KUKA KRL program: MASTER_MESA_A.src, MASTER_MESA_A.dat

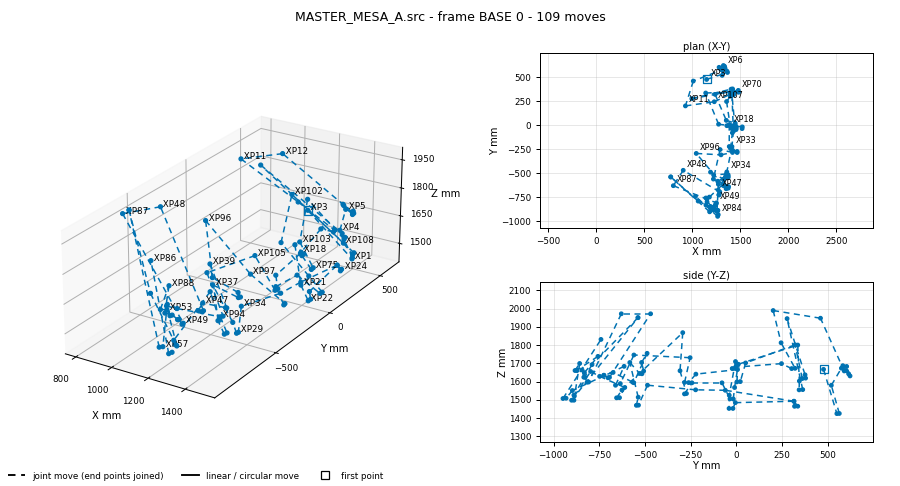
[picture p0: tool path of MASTER_MESA_A.src in frame BASE 0, 109 of 111 moves have a stored position in this frame; points joined in program order, loops and branches not executed]
--- MASTER_MESA_A.src ---
&ACCESS RVP
&REL 294
&PARAM EDITMASK = *
&PARAM TEMPLATE = C:\KRC\Roboter\Template\vorgabe
&PARAM DISKPATH = KRC:\R1\Program\Solda
DEF MASTER_MESA_A( )
;FOLD INI;%{PE}
  ;FOLD BASISTECH INI
    GLOBAL INTERRUPT DECL 3 WHEN $STOPMESS==TRUE DO IR_STOPM ( )
    INTERRUPT ON 3
    BAS (#INITMOV,0 )
  ;ENDFOLD (BASISTECH INI)
  ;FOLD USER INI
    ;Make your modifications here

  ;ENDFOLD (USER INI)
;ENDFOLD (INI)
LOOP
;FOLD PTP HOME Vel=100 % DEFAULT;%{PE}%R 8.3.48,%MKUKATPBASIS,%CMOVE,%VPTP,%P 1:PTP, 2:HOME, 3:, 5:100, 7:DEFAULT
$BWDSTART=FALSE
PDAT_ACT=PDEFAULT
FDAT_ACT=FHOME
BAS(#PTP_PARAMS,100)
$H_POS=XHOME
PTP XHOME
;ENDFOLD

;FOLD PTP P3 Vel=100 % PDAT3 Tool[1]:TOCH Base[0];%{PE}%R 8.3.48,%MKUKATPBASIS,%CMOVE,%VPTP,%P 1:PTP, 2:P3, 3:, 5:100, 7:PDAT3
$BWDSTART=FALSE
PDAT_ACT=PPDAT3
FDAT_ACT=FP3
BAS(#PTP_PARAMS,100)
PTP XP3
;ENDFOLD
;FOLD ; CORDAO 1;%{PE}%R 8.3.48,%MKUKATPBASIS,%CCOMMENT,%VNORMAL,%P 2:CORDAO 1
;ENDFOLD
;FOLD ARCON WDAT1 PTP P1 Vel=30 % PDAT2 Tool[1]:TOCH Base[0] ;%{PE}
;FOLD Parameters ;%{h}
;Params IlfProvider=kukaroboter.arctech.arconptp; Kuka.PointName=P1; Kuka.BlendingEnabled=False; Kuka.MoveDataPtpName=PDAT2; Kuka.VelocityPtp=30; Kuka.MovementParameterFieldEnabled=True; ArcTech.WdatVarName=WDAT1; ArcTech.SeamName=
;ENDFOLD
$BWDSTART = FALSE
PDAT_ACT = PPDAT2
FDAT_ACT = FP1
BAS(#PTP_PARAMS, 30.0)
TRIGGER WHEN DISTANCE = 1 DELAY = ATBg_PreDefinitionTime DO Arc_DefineStrikeParams(3, AS_WDAT1) PRIO = -1
Arc_DefineCpPattern(#OffInAdvance, WV_WDAT1, TRUE)
PTP XP1
Arc_On(1, AS_WDAT1, ATBg_StartErrSetField[1], AW_WDAT1, WV_WDAT1, ATBg_WeldErrSetField[1], #StdArcOn, " ")
Arc_DefineCpPattern(#OnInAdvance, WV_WDAT1, TRUE)
;ENDFOLD
;FOLD ARCOFF WDAT2 LIN P2 CPDAT2 Tool[1]:TOCH Base[0] ;%{PE}
;FOLD Parameters ;%{h}
;Params IlfProvider=kukaroboter.arctech.arcofflin; Kuka.PointName=P2; Kuka.BlendingEnabled=False; Kuka.MoveDataName=CPDAT2;  Kuka.MovementParameterFieldEnabled=True; ArcTech.WdatVarName=WDAT2
;ENDFOLD
$BWDSTART = FALSE
LDAT_ACT = LCPDAT2
FDAT_ACT = FP2
BAS(#CP_PARAMS, ATBg_BAS_VELDefinition)
LIN XP2
Arc_Off(1, AC_WDAT2)
;ENDFOLD
;FOLD PTP P4 Vel=100 % PDAT4 Tool[1]:TOCH Base[0];%{PE}%R 8.3.48,%MKUKATPBASIS,%CMOVE,%VPTP,%P 1:PTP, 2:P4, 3:, 5:100, 7:PDAT4
$BWDSTART=FALSE
PDAT_ACT=PPDAT4
FDAT_ACT=FP4
BAS(#PTP_PARAMS,100)
PTP XP4
;ENDFOLD
;FOLD PTP P5 Vel=100 % PDAT5 Tool[1]:TOCH Base[0];%{PE}%R 8.3.48,%MKUKATPBASIS,%CMOVE,%VPTP,%P 1:PTP, 2:P5, 3:, 5:100, 7:PDAT5
$BWDSTART=FALSE
PDAT_ACT=PPDAT5
FDAT_ACT=FP5
BAS(#PTP_PARAMS,100)
PTP XP5
;ENDFOLD
;FOLD ; CORDAO 2;%{PE}%R 8.3.48,%MKUKATPBASIS,%CCOMMENT,%VNORMAL,%P 2:CORDAO 2
;ENDFOLD
;FOLD ARCON WDAT3 PTP P6 Vel=30 % PDAT6 Tool[1]:TOCH Base[0] ;%{PE}
;FOLD Parameters ;%{h}
;Params IlfProvider=kukaroboter.arctech.arconptp; Kuka.PointName=P6; Kuka.BlendingEnabled=False; Kuka.MoveDataPtpName=PDAT6; Kuka.VelocityPtp=30; Kuka.MovementParameterFieldEnabled=True; ArcTech.WdatVarName=WDAT3; ArcTech.SeamName=
;ENDFOLD
$BWDSTART = FALSE
PDAT_ACT = PPDAT6
FDAT_ACT = FP6
BAS(#PTP_PARAMS, 30.0)
TRIGGER WHEN DISTANCE = 1 DELAY = ATBg_PreDefinitionTime DO Arc_DefineStrikeParams(3, AS_WDAT3) PRIO = -1
Arc_DefineCpPattern(#OffInAdvance, WV_WDAT3, TRUE)
PTP XP6
Arc_On(1, AS_WDAT3, ATBg_StartErrSetField[1], AW_WDAT3, WV_WDAT3, ATBg_WeldErrSetField[1], #StdArcOn, " ")
Arc_DefineCpPattern(#OnInAdvance, WV_WDAT3, TRUE)
;ENDFOLD
;FOLD ARCOFF WDAT4 LIN P7 CPDAT3 Tool[1]:TOCH Base[0] ;%{PE}
;FOLD Parameters ;%{h}
;Params IlfProvider=kukaroboter.arctech.arcofflin; Kuka.PointName=P7; Kuka.BlendingEnabled=False; Kuka.MoveDataName=CPDAT3;  Kuka.MovementParameterFieldEnabled=True; ArcTech.WdatVarName=WDAT4
;ENDFOLD
$BWDSTART = FALSE
LDAT_ACT = LCPDAT3
FDAT_ACT = FP7
BAS(#CP_PARAMS, ATBg_BAS_VELDefinition)
LIN XP7
Arc_Off(1, AC_WDAT4)
;ENDFOLD
;FOLD PTP P8 Vel=100 % PDAT7 Tool[1]:TOCH Base[0];%{PE}%R 8.3.48,%MKUKATPBASIS,%CMOVE,%VPTP,%P 1:PTP, 2:P8, 3:, 5:100, 7:PDAT7
$BWDSTART=FALSE
PDAT_ACT=PPDAT7
FDAT_ACT=FP8
BAS(#PTP_PARAMS,100)
PTP XP8
;ENDFOLD
;FOLD PTP P13 Vel=100 % PDAT11 Tool[1]:TOCH Base[0];%{PE}%R 8.3.48,%MKUKATPBASIS,%CMOVE,%VPTP,%P 1:PTP, 2:P13, 3:, 5:100, 7:PDAT11
$BWDSTART=FALSE
PDAT_ACT=PPDAT11
FDAT_ACT=FP13
BAS(#PTP_PARAMS,100)
PTP XP13
;ENDFOLD
;FOLD ; CORDAO 3;%{PE}%R 8.3.48,%MKUKATPBASIS,%CCOMMENT,%VNORMAL,%P 2:CORDAO 3
;ENDFOLD
;FOLD ARCON WDAT5 PTP P9 Vel=30 % PDAT8 Tool[1]:TOCH Base[0] ;%{PE}
;FOLD Parameters ;%{h}
;Params IlfProvider=kukaroboter.arctech.arconptp; Kuka.PointName=P9; Kuka.BlendingEnabled=False; Kuka.MoveDataPtpName=PDAT8; Kuka.VelocityPtp=30; Kuka.MovementParameterFieldEnabled=True; ArcTech.WdatVarName=WDAT5; ArcTech.SeamName=
;ENDFOLD
$BWDSTART = FALSE
PDAT_ACT = PPDAT8
FDAT_ACT = FP9
BAS(#PTP_PARAMS, 30.0)
TRIGGER WHEN DISTANCE = 1 DELAY = ATBg_PreDefinitionTime DO Arc_DefineStrikeParams(3, AS_WDAT5) PRIO = -1
Arc_DefineCpPattern(#OffInAdvance, WV_WDAT5, TRUE)
PTP XP9
Arc_On(1, AS_WDAT5, ATBg_StartErrSetField[1], AW_WDAT5, WV_WDAT5, ATBg_WeldErrSetField[1], #StdArcOn, " ")
Arc_DefineCpPattern(#OnInAdvance, WV_WDAT5, TRUE)
;ENDFOLD
;FOLD ARCOFF WDAT6 LIN P10 CPDAT4 Tool[1]:TOCH Base[0] ;%{PE}
;FOLD Parameters ;%{h}
;Params IlfProvider=kukaroboter.arctech.arcofflin; Kuka.PointName=P10; Kuka.BlendingEnabled=False; Kuka.MoveDataName=CPDAT4;  Kuka.MovementParameterFieldEnabled=True; ArcTech.WdatVarName=WDAT6
;ENDFOLD
$BWDSTART = FALSE
LDAT_ACT = LCPDAT4
FDAT_ACT = FP10
BAS(#CP_PARAMS, ATBg_BAS_VELDefinition)
LIN XP10
Arc_Off(1, AC_WDAT6)
;ENDFOLD
;FOLD PTP P12 Vel=100 % PDAT10 Tool[1]:TOCH Base[0];%{PE}%R 8.3.48,%MKUKATPBASIS,%CMOVE,%VPTP,%P 1:PTP, 2:P12, 3:, 5:100, 7:PDAT10
$BWDSTART=FALSE
PDAT_ACT=PPDAT10
FDAT_ACT=FP12
BAS(#PTP_PARAMS,100)
PTP XP12
;ENDFOLD
;FOLD PTP P11 Vel=100 % PDAT9 Tool[1]:TOCH Base[0];%{PE}%R 8.3.48,%MKUKATPBASIS,%CMOVE,%VPTP,%P 1:PTP, 2:P11, 3:, 5:100, 7:PDAT9
$BWDSTART=FALSE
PDAT_ACT=PPDAT9
FDAT_ACT=FP11
BAS(#PTP_PARAMS,100)
PTP XP11
;ENDFOLD
;FOLD PTP P107 Vel=100 % PDAT83 Tool[1]:TOCH Base[0];%{PE}%R 8.3.48,%MKUKATPBASIS,%CMOVE,%VPTP,%P 1:PTP, 2:P107, 3:, 5:100, 7:PDAT83
$BWDSTART=FALSE
PDAT_ACT=PPDAT83
FDAT_ACT=FP107
BAS(#PTP_PARAMS,100)
PTP XP107
;ENDFOLD
;FOLD ; CORDAO 4;%{PE}%R 8.3.48,%MKUKATPBASIS,%CCOMMENT,%VNORMAL,%P 2:CORDAO 4
;ENDFOLD
;FOLD ARCON WDAT7 PTP P14 Vel=30 % PDAT12 Tool[1]:TOCH Base[0] ;%{PE}
;FOLD Parameters ;%{h}
;Params IlfProvider=kukaroboter.arctech.arconptp; Kuka.PointName=P14; Kuka.BlendingEnabled=False; Kuka.MoveDataPtpName=PDAT12; Kuka.VelocityPtp=30; Kuka.MovementParameterFieldEnabled=True; ArcTech.WdatVarName=WDAT7; ArcTech.SeamName=
;ENDFOLD
$BWDSTART = FALSE
PDAT_ACT = PPDAT12
FDAT_ACT = FP14
BAS(#PTP_PARAMS, 30.0)
TRIGGER WHEN DISTANCE = 1 DELAY = ATBg_PreDefinitionTime DO Arc_DefineStrikeParams(3, AS_WDAT7) PRIO = -1
Arc_DefineCpPattern(#OffInAdvance, WV_WDAT7, TRUE)
PTP XP14
Arc_On(1, AS_WDAT7, ATBg_StartErrSetField[1], AW_WDAT7, WV_WDAT7, ATBg_WeldErrSetField[1], #StdArcOn, " ")
Arc_DefineCpPattern(#OnInAdvance, WV_WDAT7, TRUE)
;ENDFOLD
;FOLD ARCOFF WDAT8 LIN P15 CPDAT5 Tool[1]:TOCH Base[0] ;%{PE}
;FOLD Parameters ;%{h}
;Params IlfProvider=kukaroboter.arctech.arcofflin; Kuka.PointName=P15; Kuka.BlendingEnabled=False; Kuka.MoveDataName=CPDAT5;  Kuka.MovementParameterFieldEnabled=True; ArcTech.WdatVarName=WDAT8
;ENDFOLD
$BWDSTART = FALSE
LDAT_ACT = LCPDAT5
FDAT_ACT = FP15
BAS(#CP_PARAMS, ATBg_BAS_VELDefinition)
LIN XP15
Arc_Off(1, AC_WDAT8)
;ENDFOLD
;FOLD PTP P19 Vel=100 % PDAT15 Tool[1]:TOCH Base[0];%{PE}%R 8.3.48,%MKUKATPBASIS,%CMOVE,%VPTP,%P 1:PTP, 2:P19, 3:, 5:100, 7:PDAT15
$BWDSTART=FALSE
PDAT_ACT=PPDAT15
FDAT_ACT=FP19
BAS(#PTP_PARAMS,100)
PTP XP19
;ENDFOLD
;FOLD PTP P18 Vel=100 % PDAT14 Tool[1]:TOCH Base[0];%{PE}%R 8.3.48,%MKUKATPBASIS,%CMOVE,%VPTP,%P 1:PTP, 2:P18, 3:, 5:100, 7:PDAT14
$BWDSTART=FALSE
PDAT_ACT=PPDAT14
FDAT_ACT=FP18
BAS(#PTP_PARAMS,100)
PTP XP18
;ENDFOLD
;FOLD ; CORDAO 5;%{PE}%R 8.3.48,%MKUKATPBASIS,%CCOMMENT,%VNORMAL,%P 2:CORDAO 5
;ENDFOLD
;FOLD ARCON WDAT9 PTP P16 Vel=31 % PDAT13 Tool[1]:TOCH Base[0] ;%{PE}
;FOLD Parameters ;%{h}
;Params IlfProvider=kukaroboter.arctech.arconptp; Kuka.PointName=P16; Kuka.BlendingEnabled=False; Kuka.MoveDataPtpName=PDAT13; Kuka.VelocityPtp=31; Kuka.MovementParameterFieldEnabled=True; ArcTech.WdatVarName=WDAT9; ArcTech.SeamName=
;ENDFOLD
$BWDSTART = FALSE
PDAT_ACT = PPDAT13
FDAT_ACT = FP16
BAS(#PTP_PARAMS, 31.0)
TRIGGER WHEN DISTANCE = 1 DELAY = ATBg_PreDefinitionTime DO Arc_DefineStrikeParams(3, AS_WDAT9) PRIO = -1
Arc_DefineCpPattern(#OffInAdvance, WV_WDAT9, TRUE)
PTP XP16
Arc_On(1, AS_WDAT9, ATBg_StartErrSetField[1], AW_WDAT9, WV_WDAT9, ATBg_WeldErrSetField[1], #StdArcOn, " ")
Arc_DefineCpPattern(#OnInAdvance, WV_WDAT9, TRUE)
;ENDFOLD
;FOLD ARCOFF WDAT10 LIN P17 CPDAT6 Tool[1]:TOCH Base[0] ;%{PE}
;FOLD Parameters ;%{h}
;Params IlfProvider=kukaroboter.arctech.arcofflin; Kuka.PointName=P17; Kuka.BlendingEnabled=False; Kuka.MoveDataName=CPDAT6;  Kuka.MovementParameterFieldEnabled=True; ArcTech.WdatVarName=WDAT10
;ENDFOLD
$BWDSTART = FALSE
LDAT_ACT = LCPDAT6
FDAT_ACT = FP17
BAS(#CP_PARAMS, ATBg_BAS_VELDefinition)
LIN XP17
Arc_Off(1, AC_WDAT10)
;ENDFOLD
;FOLD PTP P20 Vel=100 % PDAT16 Tool[1]:TOCH Base[0];%{PE}%R 8.3.48,%MKUKATPBASIS,%CMOVE,%VPTP,%P 1:PTP, 2:P20, 3:, 5:100, 7:PDAT16
$BWDSTART=FALSE
PDAT_ACT=PPDAT16
FDAT_ACT=FP20
BAS(#PTP_PARAMS,100)
PTP XP20
;ENDFOLD
;FOLD PTP P21 Vel=100 % PDAT17 Tool[1]:TOCH Base[0];%{PE}%R 8.3.48,%MKUKATPBASIS,%CMOVE,%VPTP,%P 1:PTP, 2:P21, 3:, 5:100, 7:PDAT17
$BWDSTART=FALSE
PDAT_ACT=PPDAT17
FDAT_ACT=FP21
BAS(#PTP_PARAMS,100)
PTP XP21
;ENDFOLD
;FOLD ; CORDAO 6;%{PE}%R 8.3.48,%MKUKATPBASIS,%CCOMMENT,%VNORMAL,%P 2:CORDAO 6
;ENDFOLD
;FOLD ARCON WDAT11 PTP P22 Vel=30 % PDAT18 Tool[1]:TOCH Base[0] ;%{PE}
;FOLD Parameters ;%{h}
;Params IlfProvider=kukaroboter.arctech.arconptp; Kuka.PointName=P22; Kuka.BlendingEnabled=False; Kuka.MoveDataPtpName=PDAT18; Kuka.VelocityPtp=30; Kuka.MovementParameterFieldEnabled=True; ArcTech.WdatVarName=WDAT11; ArcTech.SeamName=
;ENDFOLD
$BWDSTART = FALSE
PDAT_ACT = PPDAT18
FDAT_ACT = FP22
BAS(#PTP_PARAMS, 30.0)
TRIGGER WHEN DISTANCE = 1 DELAY = ATBg_PreDefinitionTime DO Arc_DefineStrikeParams(3, AS_WDAT11) PRIO = -1
Arc_DefineCpPattern(#OffInAdvance, WV_WDAT11, TRUE)
PTP XP22
Arc_On(1, AS_WDAT11, ATBg_StartErrSetField[1], AW_WDAT11, WV_WDAT11, ATBg_WeldErrSetField[1], #StdArcOn, " ")
Arc_DefineCpPattern(#OnInAdvance, WV_WDAT11, TRUE)
;ENDFOLD
;FOLD ARCOFF WDAT12 LIN P23 CPDAT7 Tool[1]:TOCH Base[0] ;%{PE}
;FOLD Parameters ;%{h}
;Params IlfProvider=kukaroboter.arctech.arcofflin; Kuka.PointName=P23; Kuka.BlendingEnabled=False; Kuka.MoveDataName=CPDAT7;  Kuka.MovementParameterFieldEnabled=True; ArcTech.WdatVarName=WDAT12
;ENDFOLD
$BWDSTART = FALSE
LDAT_ACT = LCPDAT7
FDAT_ACT = FP23
BAS(#CP_PARAMS, ATBg_BAS_VELDefinition)
LIN XP23
Arc_Off(1, AC_WDAT12)
;ENDFOLD
;FOLD PTP P28 Vel=100 % PDAT22 Tool[1]:TOCH Base[0];%{PE}%R 8.3.48,%MKUKATPBASIS,%CMOVE,%VPTP,%P 1:PTP, 2:P28, 3:, 5:100, 7:PDAT22
$BWDSTART=FALSE
PDAT_ACT=PPDAT22
FDAT_ACT=FP28
BAS(#PTP_PARAMS,100)
PTP XP28
;ENDFOLD
;FOLD PTP P27 Vel=100 % PDAT21 Tool[1]:TOCH Base[0];%{PE}%R 8.3.48,%MKUKATPBASIS,%CMOVE,%VPTP,%P 1:PTP, 2:P27, 3:, 5:100, 7:PDAT21
$BWDSTART=FALSE
PDAT_ACT=PPDAT21
FDAT_ACT=FP27
BAS(#PTP_PARAMS,100)
PTP XP27
;ENDFOLD
;FOLD ; CORDAO 7;%{PE}%R 8.3.48,%MKUKATPBASIS,%CCOMMENT,%VNORMAL,%P 2:CORDAO 7
;ENDFOLD
;FOLD ARCON WDAT13 PTP P24 Vel=30 % PDAT19 Tool[1]:TOCH Base[0] ;%{PE}
;FOLD Parameters ;%{h}
;Params IlfProvider=kukaroboter.arctech.arconptp; Kuka.PointName=P24; Kuka.BlendingEnabled=False; Kuka.MoveDataPtpName=PDAT19; Kuka.VelocityPtp=30; Kuka.MovementParameterFieldEnabled=True; ArcTech.WdatVarName=WDAT13; ArcTech.SeamName=
;ENDFOLD
$BWDSTART = FALSE
PDAT_ACT = PPDAT19
FDAT_ACT = FP24
BAS(#PTP_PARAMS, 30.0)
TRIGGER WHEN DISTANCE = 1 DELAY = ATBg_PreDefinitionTime DO Arc_DefineStrikeParams(3, AS_WDAT13) PRIO = -1
Arc_DefineCpPattern(#OffInAdvance, WV_WDAT13, TRUE)
PTP XP24
Arc_On(1, AS_WDAT13, ATBg_StartErrSetField[1], AW_WDAT13, WV_WDAT13, ATBg_WeldErrSetField[1], #StdArcOn, " ")
Arc_DefineCpPattern(#OnInAdvance, WV_WDAT13, TRUE)
;ENDFOLD
;FOLD ARCOFF WDAT14 LIN P25 CPDAT8 Tool[1]:TOCH Base[0] ;%{PE}
;FOLD Parameters ;%{h}
;Params IlfProvider=kukaroboter.arctech.arcofflin; Kuka.PointName=P25; Kuka.BlendingEnabled=False; Kuka.MoveDataName=CPDAT8;  Kuka.MovementParameterFieldEnabled=True; ArcTech.WdatVarName=WDAT14
;ENDFOLD
$BWDSTART = FALSE
LDAT_ACT = LCPDAT8
FDAT_ACT = FP25
BAS(#CP_PARAMS, ATBg_BAS_VELDefinition)
LIN XP25
Arc_Off(1, AC_WDAT14)
;ENDFOLD
;FOLD PTP P26 Vel=100 % PDAT20 Tool[1]:TOCH Base[0];%{PE}%R 8.3.48,%MKUKATPBASIS,%CMOVE,%VPTP,%P 1:PTP, 2:P26, 3:, 5:100, 7:PDAT20
$BWDSTART=FALSE
PDAT_ACT=PPDAT20
FDAT_ACT=FP26
BAS(#PTP_PARAMS,100)
PTP XP26
;ENDFOLD
;FOLD PTP P32 Vel=100 % PDAT25 Tool[1]:TOCH Base[0];%{PE}%R 8.3.48,%MKUKATPBASIS,%CMOVE,%VPTP,%P 1:PTP, 2:P32, 3:, 5:100, 7:PDAT25
$BWDSTART=FALSE
PDAT_ACT=PPDAT25
FDAT_ACT=FP32
BAS(#PTP_PARAMS,100)
PTP XP32
;ENDFOLD
;FOLD PTP P33 Vel=100 % PDAT26 Tool[1]:TOCH Base[0];%{PE}%R 8.3.48,%MKUKATPBASIS,%CMOVE,%VPTP,%P 1:PTP, 2:P33, 3:, 5:100, 7:PDAT26
$BWDSTART=FALSE
PDAT_ACT=PPDAT26
FDAT_ACT=FP33
BAS(#PTP_PARAMS,100)
PTP XP33
;ENDFOLD
;FOLD PTP P34 Vel=100 % PDAT27 Tool[1]:TOCH Base[0];%{PE}%R 8.3.48,%MKUKATPBASIS,%CMOVE,%VPTP,%P 1:PTP, 2:P34, 3:, 5:100, 7:PDAT27
$BWDSTART=FALSE
PDAT_ACT=PPDAT27
FDAT_ACT=FP34
BAS(#PTP_PARAMS,100)
PTP XP34
;ENDFOLD
;FOLD ; CORDAO 8;%{PE}%R 8.3.48,%MKUKATPBASIS,%CCOMMENT,%VNORMAL,%P 2:CORDAO 8
;ENDFOLD
;FOLD ARCON WDAT15 PTP P29 Vel=30 % PDAT23 Tool[1]:TOCH Base[0] ;%{PE}
;FOLD Parameters ;%{h}
;Params IlfProvider=kukaroboter.arctech.arconptp; Kuka.PointName=P29; Kuka.BlendingEnabled=False; Kuka.MoveDataPtpName=PDAT23; Kuka.VelocityPtp=30; Kuka.MovementParameterFieldEnabled=True; ArcTech.WdatVarName=WDAT15; ArcTech.SeamName=
;ENDFOLD
$BWDSTART = FALSE
PDAT_ACT = PPDAT23
FDAT_ACT = FP29
BAS(#PTP_PARAMS, 30.0)
TRIGGER WHEN DISTANCE = 1 DELAY = ATBg_PreDefinitionTime DO Arc_DefineStrikeParams(3, AS_WDAT15) PRIO = -1
Arc_DefineCpPattern(#OffInAdvance, WV_WDAT15, TRUE)
PTP XP29
Arc_On(1, AS_WDAT15, ATBg_StartErrSetField[1], AW_WDAT15, WV_WDAT15, ATBg_WeldErrSetField[1], #StdArcOn, " ")
Arc_DefineCpPattern(#OnInAdvance, WV_WDAT15, TRUE)
;ENDFOLD
;FOLD ARCOFF WDAT16 LIN P30 CPDAT9 Tool[1]:TOCH Base[0] ;%{PE}
;FOLD Parameters ;%{h}
;Params IlfProvider=kukaroboter.arctech.arcofflin; Kuka.PointName=P30; Kuka.BlendingEnabled=False; Kuka.MoveDataName=CPDAT9;  Kuka.MovementParameterFieldEnabled=True; ArcTech.WdatVarName=WDAT16
;ENDFOLD
$BWDSTART = FALSE
LDAT_ACT = LCPDAT9
FDAT_ACT = FP30
BAS(#CP_PARAMS, ATBg_BAS_VELDefinition)
LIN XP30
Arc_Off(1, AC_WDAT16)
;ENDFOLD
;FOLD PTP P31 Vel=100 % PDAT24 Tool[1]:TOCH Base[0];%{PE}%R 8.3.48,%MKUKATPBASIS,%CMOVE,%VPTP,%P 1:PTP, 2:P31, 3:, 5:100, 7:PDAT24
$BWDSTART=FALSE
PDAT_ACT=PPDAT24
FDAT_ACT=FP31
BAS(#PTP_PARAMS,100)
PTP XP31
;ENDFOLD
;FOLD PTP P37 Vel=100 % PDAT29 Tool[1]:TOCH Base[0];%{PE}%R 8.3.48,%MKUKATPBASIS,%CMOVE,%VPTP,%P 1:PTP, 2:P37, 3:, 5:100, 7:PDAT29
$BWDSTART=FALSE
PDAT_ACT=PPDAT29
FDAT_ACT=FP37
BAS(#PTP_PARAMS,100)
PTP XP37
;ENDFOLD
;FOLD ; CORDAO 9;%{PE}%R 8.3.48,%MKUKATPBASIS,%CCOMMENT,%VNORMAL,%P 2:CORDAO 9
;ENDFOLD
;FOLD ARCON WDAT17 PTP P35 Vel=30 % PDAT28 Tool[1]:TOCH Base[0] ;%{PE}
;FOLD Parameters ;%{h}
;Params IlfProvider=kukaroboter.arctech.arconptp; Kuka.PointName=P35; Kuka.BlendingEnabled=False; Kuka.MoveDataPtpName=PDAT28; Kuka.VelocityPtp=30; Kuka.MovementParameterFieldEnabled=True; ArcTech.WdatVarName=WDAT17; ArcTech.SeamName=
;ENDFOLD
$BWDSTART = FALSE
PDAT_ACT = PPDAT28
FDAT_ACT = FP35
BAS(#PTP_PARAMS, 30.0)
TRIGGER WHEN DISTANCE = 1 DELAY = ATBg_PreDefinitionTime DO Arc_DefineStrikeParams(3, AS_WDAT17) PRIO = -1
Arc_DefineCpPattern(#OffInAdvance, WV_WDAT17, TRUE)
PTP XP35
Arc_On(1, AS_WDAT17, ATBg_StartErrSetField[1], AW_WDAT17, WV_WDAT17, ATBg_WeldErrSetField[1], #StdArcOn, " ")
Arc_DefineCpPattern(#OnInAdvance, WV_WDAT17, TRUE)
;ENDFOLD
;FOLD ARCOFF WDAT18 LIN P36 CPDAT10 Tool[1]:TOCH Base[0] ;%{PE}
;FOLD Parameters ;%{h}
;Params IlfProvider=kukaroboter.arctech.arcofflin; Kuka.PointName=P36; Kuka.BlendingEnabled=False; Kuka.MoveDataName=CPDAT10;  Kuka.MovementParameterFieldEnabled=True; ArcTech.WdatVarName=WDAT18
;ENDFOLD
$BWDSTART = FALSE
LDAT_ACT = LCPDAT10
FDAT_ACT = FP36
BAS(#CP_PARAMS, ATBg_BAS_VELDefinition)
LIN XP36
Arc_Off(1, AC_WDAT18)
;ENDFOLD
;FOLD PTP P38 Vel=100 % PDAT30 Tool[1]:TOCH Base[0];%{PE}%R 8.3.48,%MKUKATPBASIS,%CMOVE,%VPTP,%P 1:PTP, 2:P38, 3:, 5:100, 7:PDAT30
$BWDSTART=FALSE
PDAT_ACT=PPDAT30
FDAT_ACT=FP38
BAS(#PTP_PARAMS,100)
PTP XP38
;ENDFOLD
;FOLD PTP P40 Vel=100 % PDAT32 Tool[1]:TOCH Base[0];%{PE}%R 8.3.48,%MKUKATPBASIS,%CMOVE,%VPTP,%P 1:PTP, 2:P40, 3:, 5:100, 7:PDAT32
$BWDSTART=FALSE
PDAT_ACT=PPDAT32
FDAT_ACT=FP40
BAS(#PTP_PARAMS,100)
PTP XP40
;ENDFOLD
;FOLD PTP P39 Vel=100 % PDAT31 Tool[1]:TOCH Base[0];%{PE}%R 8.3.48,%MKUKATPBASIS,%CMOVE,%VPTP,%P 1:PTP, 2:P39, 3:, 5:100, 7:PDAT31
$BWDSTART=FALSE
PDAT_ACT=PPDAT31
FDAT_ACT=FP39
BAS(#PTP_PARAMS,100)
PTP XP39
;ENDFOLD
;FOLD ; CORDAO 10;%{PE}%R 8.3.48,%MKUKATPBASIS,%CCOMMENT,%VNORMAL,%P 2:CORDAO 10
;ENDFOLD
;FOLD ARCON WDAT19 PTP P41 Vel=30 % PDAT33 Tool[1]:TOCH Base[0] ;%{PE}
;FOLD Parameters ;%{h}
;Params IlfProvider=kukaroboter.arctech.arconptp; Kuka.PointName=P41; Kuka.BlendingEnabled=False; Kuka.MoveDataPtpName=PDAT33; Kuka.VelocityPtp=30; Kuka.MovementParameterFieldEnabled=True; ArcTech.WdatVarName=WDAT19; ArcTech.SeamName=
;ENDFOLD
$BWDSTART = FALSE
PDAT_ACT = PPDAT33
FDAT_ACT = FP41
BAS(#PTP_PARAMS, 30.0)
TRIGGER WHEN DISTANCE = 1 DELAY = ATBg_PreDefinitionTime DO Arc_DefineStrikeParams(3, AS_WDAT19) PRIO = -1
Arc_DefineCpPattern(#OffInAdvance, WV_WDAT19, TRUE)
PTP XP41
Arc_On(1, AS_WDAT19, ATBg_StartErrSetField[1], AW_WDAT19, WV_WDAT19, ATBg_WeldErrSetField[1], #StdArcOn, " ")
Arc_DefineCpPattern(#OnInAdvance, WV_WDAT19, TRUE)
;ENDFOLD
;FOLD ARCOFF WDAT20 LIN P42 CPDAT11 Tool[1]:TOCH Base[0] ;%{PE}
;FOLD Parameters ;%{h}
;Params IlfProvider=kukaroboter.arctech.arcofflin; Kuka.PointName=P42; Kuka.BlendingEnabled=False; Kuka.MoveDataName=CPDAT11;  Kuka.MovementParameterFieldEnabled=True; ArcTech.WdatVarName=WDAT20
;ENDFOLD
$BWDSTART = FALSE
LDAT_ACT = LCPDAT11
FDAT_ACT = FP42
BAS(#CP_PARAMS, ATBg_BAS_VELDefinition)
LIN XP42
Arc_Off(1, AC_WDAT20)
;ENDFOLD
;FOLD PTP P47 Vel=100 % PDAT36 Tool[1]:TOCH Base[0];%{PE}%R 8.3.48,%MKUKATPBASIS,%CMOVE,%VPTP,%P 1:PTP, 2:P47, 3:, 5:100, 7:PDAT36
$BWDSTART=FALSE
PDAT_ACT=PPDAT36
FDAT_ACT=FP47
BAS(#PTP_PARAMS,100)
PTP XP47
;ENDFOLD
;FOLD ; CORDAO 11;%{PE}%R 8.3.48,%MKUKATPBASIS,%CCOMMENT,%VNORMAL,%P 2:CORDAO 11
;ENDFOLD
;FOLD ARCON WDAT21 PTP P43 Vel=30 % PDAT34 Tool[1]:TOCH Base[0] ;%{PE}
;FOLD Parameters ;%{h}
;Params IlfProvider=kukaroboter.arctech.arconptp; Kuka.PointName=P43; Kuka.BlendingEnabled=False; Kuka.MoveDataPtpName=PDAT34; Kuka.VelocityPtp=30; Kuka.MovementParameterFieldEnabled=True; ArcTech.WdatVarName=WDAT21; ArcTech.SeamName=
;ENDFOLD
$BWDSTART = FALSE
PDAT_ACT = PPDAT34
FDAT_ACT = FP43
BAS(#PTP_PARAMS, 30.0)
TRIGGER WHEN DISTANCE = 1 DELAY = ATBg_PreDefinitionTime DO Arc_DefineStrikeParams(3, AS_WDAT21) PRIO = -1
Arc_DefineCpPattern(#OffInAdvance, WV_WDAT21, TRUE)
PTP XP43
Arc_On(1, AS_WDAT21, ATBg_StartErrSetField[1], AW_WDAT21, WV_WDAT21, ATBg_WeldErrSetField[1], #StdArcOn, " ")
Arc_DefineCpPattern(#OnInAdvance, WV_WDAT21, TRUE)
;ENDFOLD
;FOLD ARCOFF WDAT22 LIN P44 CPDAT12 Tool[1]:TOCH Base[0] ;%{PE}
;FOLD Parameters ;%{h}
;Params IlfProvider=kukaroboter.arctech.arcofflin; Kuka.PointName=P44; Kuka.BlendingEnabled=False; Kuka.MoveDataName=CPDAT12;  Kuka.MovementParameterFieldEnabled=True; ArcTech.WdatVarName=WDAT22
;ENDFOLD
$BWDSTART = FALSE
LDAT_ACT = LCPDAT12
FDAT_ACT = FP44
BAS(#CP_PARAMS, ATBg_BAS_VELDefinition)
LIN XP44
Arc_Off(1, AC_WDAT22)
;ENDFOLD
;FOLD ; CORDAO 12;%{PE}%R 8.3.48,%MKUKATPBASIS,%CCOMMENT,%VNORMAL,%P 2:CORDAO 12
;ENDFOLD
;FOLD ARCON WDAT23 PTP P45 Vel=30 % PDAT35 Tool[1]:TOCH Base[0] ;%{PE}
;FOLD Parameters ;%{h}
;Params IlfProvider=kukaroboter.arctech.arconptp; Kuka.PointName=P45; Kuka.BlendingEnabled=False; Kuka.MoveDataPtpName=PDAT35; Kuka.VelocityPtp=30; Kuka.MovementParameterFieldEnabled=True; ArcTech.WdatVarName=WDAT23; ArcTech.SeamName=
;ENDFOLD
$BWDSTART = FALSE
PDAT_ACT = PPDAT35
FDAT_ACT = FP45
BAS(#PTP_PARAMS, 30.0)
TRIGGER WHEN DISTANCE = 1 DELAY = ATBg_PreDefinitionTime DO Arc_DefineStrikeParams(1, AS_WDAT23) PRIO = -1
Arc_DefineCpPattern(#OffInAdvance, WV_WDAT23, TRUE)
PTP XP45
Arc_On(1, AS_WDAT23, ATBg_StartErrSetField[1], AW_WDAT23, WV_WDAT23, ATBg_WeldErrSetField[1], #StdArcOn, " ")
Arc_DefineCpPattern(#OnInAdvance, WV_WDAT23, TRUE)
;ENDFOLD
;FOLD ARCOFF WDAT24 LIN P46 CPDAT13 Tool[1]:TOCH Base[0] ;%{PE}
;FOLD Parameters ;%{h}
;Params IlfProvider=kukaroboter.arctech.arcofflin; Kuka.PointName=P46; Kuka.BlendingEnabled=False; Kuka.MoveDataName=CPDAT13;  Kuka.MovementParameterFieldEnabled=True; ArcTech.WdatVarName=WDAT24
;ENDFOLD
$BWDSTART = FALSE
LDAT_ACT = LCPDAT13
FDAT_ACT = FP46
BAS(#CP_PARAMS, ATBg_BAS_VELDefinition)
LIN XP46
Arc_Off(1, AC_WDAT24)
;ENDFOLD
;FOLD PTP P48 Vel=100 % PDAT37 Tool[1]:TOCH Base[0];%{PE}%R 8.3.48,%MKUKATPBASIS,%CMOVE,%VPTP,%P 1:PTP, 2:P48, 3:, 5:100, 7:PDAT37
$BWDSTART=FALSE
PDAT_ACT=PPDAT37
FDAT_ACT=FP48
BAS(#PTP_PARAMS,100)
PTP XP48
;ENDFOLD
;FOLD PTP P87 Vel=100 % PDAT62 Tool[1]:TOCH Base[0];%{PE}%R 8.3.48,%MKUKATPBASIS,%CMOVE,%VPTP,%P 1:PTP, 2:P87, 3:, 5:100, 7:PDAT62
$BWDSTART=FALSE
PDAT_ACT=PPDAT62
FDAT_ACT=FP87
BAS(#PTP_PARAMS,100)
PTP XP87
;ENDFOLD
;FOLD ; CORDAO 13;%{PE}%R 8.3.48,%MKUKATPBASIS,%CCOMMENT,%VNORMAL,%P 2:CORDAO 13
;ENDFOLD
;FOLD ARCON WDAT25 PTP P49 Vel=30 % PDAT38 Tool[1]:TOCH Base[0] ;%{PE}
;FOLD Parameters ;%{h}
;Params IlfProvider=kukaroboter.arctech.arconptp; Kuka.PointName=P49; Kuka.BlendingEnabled=False; Kuka.MoveDataPtpName=PDAT38; Kuka.VelocityPtp=30; Kuka.MovementParameterFieldEnabled=True; ArcTech.WdatVarName=WDAT25; ArcTech.SeamName=
;ENDFOLD
$BWDSTART = FALSE
PDAT_ACT = PPDAT38
FDAT_ACT = FP49
BAS(#PTP_PARAMS, 30.0)
TRIGGER WHEN DISTANCE = 1 DELAY = ATBg_PreDefinitionTime DO Arc_DefineStrikeParams(3, AS_WDAT25) PRIO = -1
Arc_DefineCpPattern(#OffInAdvance, WV_WDAT25, TRUE)
PTP XP49
Arc_On(1, AS_WDAT25, ATBg_StartErrSetField[1], AW_WDAT25, WV_WDAT25, ATBg_WeldErrSetField[1], #StdArcOn, " ")
Arc_DefineCpPattern(#OnInAdvance, WV_WDAT25, TRUE)
;ENDFOLD
;FOLD ARCOFF WDAT26 LIN P50 CPDAT14 Tool[1]:TOCH Base[0] ;%{PE}
;FOLD Parameters ;%{h}
;Params IlfProvider=kukaroboter.arctech.arcofflin; Kuka.PointName=P50; Kuka.BlendingEnabled=False; Kuka.MoveDataName=CPDAT14;  Kuka.MovementParameterFieldEnabled=True; ArcTech.WdatVarName=WDAT26
;ENDFOLD
$BWDSTART = FALSE
LDAT_ACT = LCPDAT14
FDAT_ACT = FP50
BAS(#CP_PARAMS, ATBg_BAS_VELDefinition)
LIN XP50
Arc_Off(1, AC_WDAT26)
;ENDFOLD
;FOLD ; CORDAO 14;%{PE}%R 8.3.48,%MKUKATPBASIS,%CCOMMENT,%VNORMAL,%P 2:CORDAO 14
;ENDFOLD
;FOLD ARCON WDAT27 PTP P51 Vel=30 % PDAT39 Tool[1]:TOCH Base[0] ;%{PE}
;FOLD Parameters ;%{h}
;Params IlfProvider=kukaroboter.arctech.arconptp; Kuka.PointName=P51; Kuka.BlendingEnabled=False; Kuka.MoveDataPtpName=PDAT39; Kuka.VelocityPtp=30; Kuka.MovementParameterFieldEnabled=True; ArcTech.WdatVarName=WDAT27; ArcTech.SeamName=
;ENDFOLD
$BWDSTART = FALSE
PDAT_ACT = PPDAT39
FDAT_ACT = FP51
BAS(#PTP_PARAMS, 30.0)
TRIGGER WHEN DISTANCE = 1 DELAY = ATBg_PreDefinitionTime DO Arc_DefineStrikeParams(3, AS_WDAT27) PRIO = -1
Arc_DefineCpPattern(#OffInAdvance, WV_WDAT27, TRUE)
PTP XP51
Arc_On(1, AS_WDAT27, ATBg_StartErrSetField[1], AW_WDAT27, WV_WDAT27, ATBg_WeldErrSetField[1], #StdArcOn, " ")
Arc_DefineCpPattern(#OnInAdvance, WV_WDAT27, TRUE)
;ENDFOLD
;FOLD ARCOFF WDAT28 LIN P52 CPDAT15 Tool[1]:TOCH Base[0] ;%{PE}
;FOLD Parameters ;%{h}
;Params IlfProvider=kukaroboter.arctech.arcofflin; Kuka.PointName=P52; Kuka.BlendingEnabled=False; Kuka.MoveDataName=CPDAT15;  Kuka.MovementParameterFieldEnabled=True; ArcTech.WdatVarName=WDAT28
;ENDFOLD
$BWDSTART = FALSE
LDAT_ACT = LCPDAT15
FDAT_ACT = FP52
BAS(#CP_PARAMS, ATBg_BAS_VELDefinition)
LIN XP52
Arc_Off(1, AC_WDAT28)
;ENDFOLD
;FOLD PTP P53 Vel=100 % PDAT40 Tool[1]:TOCH Base[0];%{PE}%R 8.3.48,%MKUKATPBASIS,%CMOVE,%VPTP,%P 1:PTP, 2:P53, 3:, 5:100, 7:PDAT40
$BWDSTART=FALSE
PDAT_ACT=PPDAT40
FDAT_ACT=FP53
BAS(#PTP_PARAMS,100)
PTP XP53
;ENDFOLD
;FOLD PTP P89 Vel=100 % PDAT64 Tool[1]:TOCH Base[0];%{PE}%R 8.3.48,%MKUKATPBASIS,%CMOVE,%VPTP,%P 1:PTP, 2:P89, 3:, 5:100, 7:PDAT64
$BWDSTART=FALSE
PDAT_ACT=PPDAT64
FDAT_ACT=FP89
BAS(#PTP_PARAMS,100)
PTP XP89
;ENDFOLD
;FOLD PTP P88 Vel=100 % PDAT63 Tool[1]:TOCH Base[0];%{PE}%R 8.3.48,%MKUKATPBASIS,%CMOVE,%VPTP,%P 1:PTP, 2:P88, 3:, 5:100, 7:PDAT63
$BWDSTART=FALSE
PDAT_ACT=PPDAT63
FDAT_ACT=FP88
BAS(#PTP_PARAMS,100)
PTP XP88
;ENDFOLD
;FOLD PTP P90 Vel=100 % PDAT65 Tool[1]:TOCH Base[0];%{PE}%R 8.3.48,%MKUKATPBASIS,%CMOVE,%VPTP,%P 1:PTP, 2:P90, 3:, 5:100, 7:PDAT65
$BWDSTART=FALSE
PDAT_ACT=PPDAT65
FDAT_ACT=FP90
BAS(#PTP_PARAMS,100)
PTP XP90
;ENDFOLD
;FOLD ; CORDAO 15;%{PE}%R 8.3.48,%MKUKATPBASIS,%CCOMMENT,%VNORMAL,%P 2:CORDAO 15
;ENDFOLD
;FOLD ARCON WDAT29 PTP P54 Vel=30 % PDAT41 Tool[1]:TOCH Base[0] ;%{PE}
;FOLD Parameters ;%{h}
;Params IlfProvider=kukaroboter.arctech.arconptp; Kuka.PointName=P54; Kuka.BlendingEnabled=False; Kuka.MoveDataPtpName=PDAT41; Kuka.VelocityPtp=30; Kuka.MovementParameterFieldEnabled=True; ArcTech.WdatVarName=WDAT29; ArcTech.SeamName=
;ENDFOLD
$BWDSTART = FALSE
PDAT_ACT = PPDAT41
FDAT_ACT = FP54
BAS(#PTP_PARAMS, 30.0)
TRIGGER WHEN DISTANCE = 1 DELAY = ATBg_PreDefinitionTime DO Arc_DefineStrikeParams(3, AS_WDAT29) PRIO = -1
Arc_DefineCpPattern(#OffInAdvance, WV_WDAT29, TRUE)
PTP XP54
Arc_On(1, AS_WDAT29, ATBg_StartErrSetField[1], AW_WDAT29, WV_WDAT29, ATBg_WeldErrSetField[1], #StdArcOn, " ")
Arc_DefineCpPattern(#OnInAdvance, WV_WDAT29, TRUE)
;ENDFOLD
;FOLD ARCOFF WDAT30 LIN P55 CPDAT16 Tool[1]:TOCH Base[0] ;%{PE}
;FOLD Parameters ;%{h}
;Params IlfProvider=kukaroboter.arctech.arcofflin; Kuka.PointName=P55; Kuka.BlendingEnabled=False; Kuka.MoveDataName=CPDAT16;  Kuka.MovementParameterFieldEnabled=True; ArcTech.WdatVarName=WDAT30
;ENDFOLD
$BWDSTART = FALSE
LDAT_ACT = LCPDAT16
FDAT_ACT = FP55
BAS(#CP_PARAMS, ATBg_BAS_VELDefinition)
LIN XP55
Arc_Off(1, AC_WDAT30)
;ENDFOLD
;FOLD PTP P56 Vel=100 % PDAT42 Tool[1]:TOCH Base[0];%{PE}%R 8.3.48,%MKUKATPBASIS,%CMOVE,%VPTP,%P 1:PTP, 2:P56, 3:, 5:100, 7:PDAT42
$BWDSTART=FALSE
PDAT_ACT=PPDAT42
FDAT_ACT=FP56
BAS(#PTP_PARAMS,100)
PTP XP56
;ENDFOLD
;FOLD ; CORDAO 16;%{PE}%R 8.3.48,%MKUKATPBASIS,%CCOMMENT,%VNORMAL,%P 2:CORDAO 16
;ENDFOLD
;FOLD ARCON WDAT31 PTP P57 Vel=30 % PDAT43 Tool[1]:TOCH Base[0] ;%{PE}
;FOLD Parameters ;%{h}
;Params IlfProvider=kukaroboter.arctech.arconptp; Kuka.PointName=P57; Kuka.BlendingEnabled=False; Kuka.MoveDataPtpName=PDAT43; Kuka.VelocityPtp=30; Kuka.MovementParameterFieldEnabled=True; ArcTech.WdatVarName=WDAT31; ArcTech.SeamName=
;ENDFOLD
$BWDSTART = FALSE
PDAT_ACT = PPDAT43
FDAT_ACT = FP57
BAS(#PTP_PARAMS, 30.0)
TRIGGER WHEN DISTANCE = 1 DELAY = ATBg_PreDefinitionTime DO Arc_DefineStrikeParams(3, AS_WDAT31) PRIO = -1
Arc_DefineCpPattern(#OffInAdvance, WV_WDAT31, TRUE)
PTP XP57
Arc_On(1, AS_WDAT31, ATBg_StartErrSetField[1], AW_WDAT31, WV_WDAT31, ATBg_WeldErrSetField[1], #StdArcOn, " ")
Arc_DefineCpPattern(#OnInAdvance, WV_WDAT31, TRUE)
;ENDFOLD
;FOLD ARCOFF WDAT32 LIN P58 CPDAT17 Tool[1]:TOCH Base[0] ;%{PE}
;FOLD Parameters ;%{h}
;Params IlfProvider=kukaroboter.arctech.arcofflin; Kuka.PointName=P58; Kuka.BlendingEnabled=False; Kuka.MoveDataName=CPDAT17;  Kuka.MovementParameterFieldEnabled=True; ArcTech.WdatVarName=WDAT32
;ENDFOLD
$BWDSTART = FALSE
LDAT_ACT = LCPDAT17
FDAT_ACT = FP58
BAS(#CP_PARAMS, ATBg_BAS_VELDefinition)
LIN XP58
Arc_Off(1, AC_WDAT32)
;ENDFOLD
;FOLD PTP P59 Vel=100 % PDAT44 Tool[1]:TOCH Base[0];%{PE}%R 8.3.48,%MKUKATPBASIS,%CMOVE,%VPTP,%P 1:PTP, 2:P59, 3:, 5:100, 7:PDAT44
$BWDSTART=FALSE
PDAT_ACT=PPDAT44
FDAT_ACT=FP59
BAS(#PTP_PARAMS,100)
PTP XP59
;ENDFOLD
;FOLD PTP P60 Vel=100 % PDAT45 Tool[1]:TOCH Base[0];%{PE}%R 8.3.48,%MKUKATPBASIS,%CMOVE,%VPTP,%P 1:PTP, 2:P60, 3:, 5:100, 7:PDAT45
$BWDSTART=FALSE
PDAT_ACT=PPDAT45
FDAT_ACT=FP60
BAS(#PTP_PARAMS,100)
PTP XP60
;ENDFOLD
;FOLD PTP P91 Vel=100 % PDAT67 Tool[1]:TOCH Base[0];%{PE}%R 8.3.48,%MKUKATPBASIS,%CMOVE,%VPTP,%P 1:PTP, 2:P91, 3:, 5:100, 7:PDAT67
$BWDSTART=FALSE
PDAT_ACT=PPDAT67
FDAT_ACT=FP91
BAS(#PTP_PARAMS,100)
PTP XP91
;ENDFOLD
;FOLD ; CORDAO 17;%{PE}%R 8.3.48,%MKUKATPBASIS,%CCOMMENT,%VNORMAL,%P 2:CORDAO 17
;ENDFOLD
;FOLD ARCON WDAT33 PTP P61 Vel=30 % PDAT66 Tool[1]:TOCH Base[0] ;%{PE}
;FOLD Parameters ;%{h}
;Params IlfProvider=kukaroboter.arctech.arconptp; Kuka.PointName=P61; Kuka.BlendingEnabled=False; Kuka.MoveDataPtpName=PDAT66; Kuka.VelocityPtp=30; Kuka.MovementParameterFieldEnabled=True; ArcTech.WdatVarName=WDAT33; ArcTech.SeamName=
;ENDFOLD
$BWDSTART = FALSE
PDAT_ACT = PPDAT66
FDAT_ACT = FP61
BAS(#PTP_PARAMS, 30.0)
TRIGGER WHEN DISTANCE = 1 DELAY = ATBg_PreDefinitionTime DO Arc_DefineStrikeParams(3, AS_WDAT33) PRIO = -1
Arc_DefineCpPattern(#OffInAdvance, WV_WDAT33, TRUE)
PTP XP61
Arc_On(1, AS_WDAT33, ATBg_StartErrSetField[1], AW_WDAT33, WV_WDAT33, ATBg_WeldErrSetField[1], #StdArcOn, " ")
Arc_DefineCpPattern(#OnInAdvance, WV_WDAT33, TRUE)
;ENDFOLD
;FOLD ARCOFF WDAT34 LIN P62 CPDAT18 Tool[1]:TOCH Base[0] ;%{PE}
;FOLD Parameters ;%{h}
;Params IlfProvider=kukaroboter.arctech.arcofflin; Kuka.PointName=P62; Kuka.BlendingEnabled=False; Kuka.MoveDataName=CPDAT18;  Kuka.MovementParameterFieldEnabled=True; ArcTech.WdatVarName=WDAT34
;ENDFOLD
$BWDSTART = FALSE
LDAT_ACT = LCPDAT18
FDAT_ACT = FP62
BAS(#CP_PARAMS, ATBg_BAS_VELDefinition)
LIN XP62
Arc_Off(1, AC_WDAT34)
;ENDFOLD
;FOLD PTP P92 Vel=100 % PDAT68 Tool[1]:TOCH Base[0];%{PE}%R 8.3.48,%MKUKATPBASIS,%CMOVE,%VPTP,%P 1:PTP, 2:P92, 3:, 5:100, 7:PDAT68
$BWDSTART=FALSE
PDAT_ACT=PPDAT68
FDAT_ACT=FP92
BAS(#PTP_PARAMS,100)
PTP XP92
;ENDFOLD
;FOLD PTP P93 Vel=100 % PDAT69 Tool[1]:TOCH Base[0];%{PE}%R 8.3.48,%MKUKATPBASIS,%CMOVE,%VPTP,%P 1:PTP, 2:P93, 3:, 5:100, 7:PDAT69
$BWDSTART=FALSE
PDAT_ACT=PPDAT69
FDAT_ACT=FP93
BAS(#PTP_PARAMS,100)
PTP XP93
;ENDFOLD
;FOLD PTP P94 Vel=100 % PDAT70 Tool[1]:TOCH Base[0];%{PE}%R 8.3.48,%MKUKATPBASIS,%CMOVE,%VPTP,%P 1:PTP, 2:P94, 3:, 5:100, 7:PDAT70
$BWDSTART=FALSE
PDAT_ACT=PPDAT70
FDAT_ACT=FP94
BAS(#PTP_PARAMS,100)
PTP XP94
;ENDFOLD
;FOLD ; CORDAO 18;%{PE}%R 8.3.48,%MKUKATPBASIS,%CCOMMENT,%VNORMAL,%P 2:CORDAO 18
;ENDFOLD
;FOLD ARCON WDAT35 PTP P63 Vel=30 % PDAT47 Tool[1]:TOCH Base[0] ;%{PE}
;FOLD Parameters ;%{h}
;Params IlfProvider=kukaroboter.arctech.arconptp; Kuka.PointName=P63; Kuka.BlendingEnabled=False; Kuka.MoveDataPtpName=PDAT47; Kuka.VelocityPtp=30; Kuka.MovementParameterFieldEnabled=True; ArcTech.WdatVarName=WDAT35; ArcTech.SeamName=
;ENDFOLD
$BWDSTART = FALSE
PDAT_ACT = PPDAT47
FDAT_ACT = FP63
BAS(#PTP_PARAMS, 30.0)
TRIGGER WHEN DISTANCE = 1 DELAY = ATBg_PreDefinitionTime DO Arc_DefineStrikeParams(3, AS_WDAT35) PRIO = -1
Arc_DefineCpPattern(#OffInAdvance, WV_WDAT35, TRUE)
PTP XP63
Arc_On(1, AS_WDAT35, ATBg_StartErrSetField[1], AW_WDAT35, WV_WDAT35, ATBg_WeldErrSetField[1], #StdArcOn, " ")
Arc_DefineCpPattern(#OnInAdvance, WV_WDAT35, TRUE)
;ENDFOLD
;FOLD ARCOFF WDAT36 LIN P64 CPDAT19 Tool[1]:TOCH Base[0] ;%{PE}
;FOLD Parameters ;%{h}
;Params IlfProvider=kukaroboter.arctech.arcofflin; Kuka.PointName=P64; Kuka.BlendingEnabled=False; Kuka.MoveDataName=CPDAT19;  Kuka.MovementParameterFieldEnabled=True; ArcTech.WdatVarName=WDAT36
;ENDFOLD
$BWDSTART = FALSE
LDAT_ACT = LCPDAT19
FDAT_ACT = FP64
BAS(#CP_PARAMS, ATBg_BAS_VELDefinition)
LIN XP64
Arc_Off(1, AC_WDAT36)
;ENDFOLD
;FOLD PTP P95 Vel=100 % PDAT71 Tool[1]:TOCH Base[0];%{PE}%R 8.3.48,%MKUKATPBASIS,%CMOVE,%VPTP,%P 1:PTP, 2:P95, 3:, 5:100, 7:PDAT71
$BWDSTART=FALSE
PDAT_ACT=PPDAT71
FDAT_ACT=FP95
BAS(#PTP_PARAMS,100)
PTP XP95
;ENDFOLD
;FOLD PTP P96 Vel=100 % PDAT72 Tool[1]:TOCH Base[0];%{PE}%R 8.3.48,%MKUKATPBASIS,%CMOVE,%VPTP,%P 1:PTP, 2:P96, 3:, 5:100, 7:PDAT72
$BWDSTART=FALSE
PDAT_ACT=PPDAT72
FDAT_ACT=FP96
BAS(#PTP_PARAMS,100)
PTP XP96
;ENDFOLD
;FOLD PTP P97 Vel=100 % PDAT73 Tool[1]:TOCH Base[0];%{PE}%R 8.3.48,%MKUKATPBASIS,%CMOVE,%VPTP,%P 1:PTP, 2:P97, 3:, 5:100, 7:PDAT73
$BWDSTART=FALSE
PDAT_ACT=PPDAT73
FDAT_ACT=FP97
BAS(#PTP_PARAMS,100)
PTP XP97
;ENDFOLD
;FOLD ; CORDAO 19;%{PE}%R 8.3.48,%MKUKATPBASIS,%CCOMMENT,%VNORMAL,%P 2:CORDAO 19
;ENDFOLD
;FOLD ARCON WDAT37 PTP P65 Vel=30 % PDAT48 Tool[1]:TOCH Base[0] ;%{PE}
;FOLD Parameters ;%{h}
;Params IlfProvider=kukaroboter.arctech.arconptp; Kuka.PointName=P65; Kuka.BlendingEnabled=False; Kuka.MoveDataPtpName=PDAT48; Kuka.VelocityPtp=30; Kuka.MovementParameterFieldEnabled=True; ArcTech.WdatVarName=WDAT37; ArcTech.SeamName=
;ENDFOLD
$BWDSTART = FALSE
PDAT_ACT = PPDAT48
FDAT_ACT = FP65
BAS(#PTP_PARAMS, 30.0)
TRIGGER WHEN DISTANCE = 1 DELAY = ATBg_PreDefinitionTime DO Arc_DefineStrikeParams(3, AS_WDAT37) PRIO = -1
Arc_DefineCpPattern(#OffInAdvance, WV_WDAT37, TRUE)
PTP XP65
Arc_On(1, AS_WDAT37, ATBg_StartErrSetField[1], AW_WDAT37, WV_WDAT37, ATBg_WeldErrSetField[1], #StdArcOn, " ")
Arc_DefineCpPattern(#OnInAdvance, WV_WDAT37, TRUE)
;ENDFOLD
;FOLD ARCOFF WDAT38 LIN P66 CPDAT20 Tool[1]:TOCH Base[0] ;%{PE}
;FOLD Parameters ;%{h}
;Params IlfProvider=kukaroboter.arctech.arcofflin; Kuka.PointName=P66; Kuka.BlendingEnabled=False; Kuka.MoveDataName=CPDAT20;  Kuka.MovementParameterFieldEnabled=True; ArcTech.WdatVarName=WDAT38
;ENDFOLD
$BWDSTART = FALSE
LDAT_ACT = LCPDAT20
FDAT_ACT = FP66
BAS(#CP_PARAMS, ATBg_BAS_VELDefinition)
LIN XP66
Arc_Off(1, AC_WDAT38)
;ENDFOLD
;FOLD PTP P98 Vel=100 % PDAT74 Tool[1]:TOCH Base[0];%{PE}%R 8.3.48,%MKUKATPBASIS,%CMOVE,%VPTP,%P 1:PTP, 2:P98, 3:, 5:100, 7:PDAT74
$BWDSTART=FALSE
PDAT_ACT=PPDAT74
FDAT_ACT=FP98
BAS(#PTP_PARAMS,100)
PTP XP98
;ENDFOLD
;FOLD PTP P99 Vel=100 % PDAT75 Tool[1]:TOCH Base[0];%{PE}%R 8.3.48,%MKUKATPBASIS,%CMOVE,%VPTP,%P 1:PTP, 2:P99, 3:, 5:100, 7:PDAT75
$BWDSTART=FALSE
PDAT_ACT=PPDAT75
FDAT_ACT=FP99
BAS(#PTP_PARAMS,100)
PTP XP99
;ENDFOLD
;FOLD ; CORDAO 20;%{PE}%R 8.3.48,%MKUKATPBASIS,%CCOMMENT,%VNORMAL,%P 2:CORDAO 20
;ENDFOLD
;FOLD ARCON WDAT39 PTP P67 Vel=30 % PDAT49 Tool[1]:TOCH Base[0] ;%{PE}
;FOLD Parameters ;%{h}
;Params IlfProvider=kukaroboter.arctech.arconptp; Kuka.PointName=P67; Kuka.BlendingEnabled=False; Kuka.MoveDataPtpName=PDAT49; Kuka.VelocityPtp=30; Kuka.MovementParameterFieldEnabled=True; ArcTech.WdatVarName=WDAT39; ArcTech.SeamName=
;ENDFOLD
$BWDSTART = FALSE
PDAT_ACT = PPDAT49
FDAT_ACT = FP67
BAS(#PTP_PARAMS, 30.0)
TRIGGER WHEN DISTANCE = 1 DELAY = ATBg_PreDefinitionTime DO Arc_DefineStrikeParams(3, AS_WDAT39) PRIO = -1
Arc_DefineCpPattern(#OffInAdvance, WV_WDAT39, TRUE)
PTP XP67
Arc_On(1, AS_WDAT39, ATBg_StartErrSetField[1], AW_WDAT39, WV_WDAT39, ATBg_WeldErrSetField[1], #StdArcOn, " ")
Arc_DefineCpPattern(#OnInAdvance, WV_WDAT39, TRUE)
;ENDFOLD
;FOLD ARCOFF WDAT40 LIN P68 CPDAT21 Tool[1]:TOCH Base[0] ;%{PE}
;FOLD Parameters ;%{h}
;Params IlfProvider=kukaroboter.arctech.arcofflin; Kuka.PointName=P68; Kuka.BlendingEnabled=False; Kuka.MoveDataName=CPDAT21;  Kuka.MovementParameterFieldEnabled=True; ArcTech.WdatVarName=WDAT40
;ENDFOLD
$BWDSTART = FALSE
LDAT_ACT = LCPDAT21
FDAT_ACT = FP68
BAS(#CP_PARAMS, ATBg_BAS_VELDefinition)
LIN XP68
Arc_Off(1, AC_WDAT40)
;ENDFOLD
;FOLD PTP P100 Vel=100 % PDAT76 Tool[1]:TOCH Base[0];%{PE}%R 8.3.48,%MKUKATPBASIS,%CMOVE,%VPTP,%P 1:PTP, 2:P100, 3:, 5:100, 7:PDAT76
$BWDSTART=FALSE
PDAT_ACT=PPDAT76
FDAT_ACT=FP100
BAS(#PTP_PARAMS,100)
PTP XP100
;ENDFOLD
;FOLD PTP P101 Vel=100 % PDAT77 Tool[1]:TOCH Base[0];%{PE}%R 8.3.48,%MKUKATPBASIS,%CMOVE,%VPTP,%P 1:PTP, 2:P101, 3:, 5:100, 7:PDAT77
$BWDSTART=FALSE
PDAT_ACT=PPDAT77
FDAT_ACT=FP101
BAS(#PTP_PARAMS,100)
PTP XP101
;ENDFOLD
;FOLD PTP P102 Vel=100 % PDAT78 Tool[1]:TOCH Base[0];%{PE}%R 8.3.48,%MKUKATPBASIS,%CMOVE,%VPTP,%P 1:PTP, 2:P102, 3:, 5:100, 7:PDAT78
$BWDSTART=FALSE
PDAT_ACT=PPDAT78
FDAT_ACT=FP102
BAS(#PTP_PARAMS,100)
PTP XP102
;ENDFOLD
;FOLD PTP P108 Vel=100 % PDAT84 Tool[1]:TOCH Base[0];%{PE}%R 8.3.48,%MKUKATPBASIS,%CMOVE,%VPTP,%P 1:PTP, 2:P108, 3:, 5:100, 7:PDAT84
$BWDSTART=FALSE
PDAT_ACT=PPDAT84
FDAT_ACT=FP108
BAS(#PTP_PARAMS,100)
PTP XP108
;ENDFOLD
;FOLD ; CORDAO 21;%{PE}%R 8.3.48,%MKUKATPBASIS,%CCOMMENT,%VNORMAL,%P 2:CORDAO 21
;ENDFOLD
;FOLD ARCON WDAT41 PTP P69 Vel=30 % PDAT50 Tool[1]:TOCH Base[0] ;%{PE}
;FOLD Parameters ;%{h}
;Params IlfProvider=kukaroboter.arctech.arconptp; Kuka.PointName=P69; Kuka.BlendingEnabled=False; Kuka.MoveDataPtpName=PDAT50; Kuka.VelocityPtp=30; Kuka.MovementParameterFieldEnabled=True; ArcTech.WdatVarName=WDAT41; ArcTech.SeamName=
;ENDFOLD
$BWDSTART = FALSE
PDAT_ACT = PPDAT50
FDAT_ACT = FP69
BAS(#PTP_PARAMS, 30.0)
TRIGGER WHEN DISTANCE = 1 DELAY = ATBg_PreDefinitionTime DO Arc_DefineStrikeParams(3, AS_WDAT41) PRIO = -1
Arc_DefineCpPattern(#OffInAdvance, WV_WDAT41, TRUE)
PTP XP69
Arc_On(1, AS_WDAT41, ATBg_StartErrSetField[1], AW_WDAT41, WV_WDAT41, ATBg_WeldErrSetField[1], #StdArcOn, " ")
Arc_DefineCpPattern(#OnInAdvance, WV_WDAT41, TRUE)
;ENDFOLD
;FOLD ARCOFF WDAT42 LIN P70 CPDAT22 Tool[1]:TOCH Base[0] ;%{PE}
;FOLD Parameters ;%{h}
;Params IlfProvider=kukaroboter.arctech.arcofflin; Kuka.PointName=P70; Kuka.BlendingEnabled=False; Kuka.MoveDataName=CPDAT22;  Kuka.MovementParameterFieldEnabled=True; ArcTech.WdatVarName=WDAT42
;ENDFOLD
$BWDSTART = FALSE
LDAT_ACT = LCPDAT22
FDAT_ACT = FP70
BAS(#CP_PARAMS, ATBg_BAS_VELDefinition)
LIN XP70
Arc_Off(1, AC_WDAT42)
;ENDFOLD
;FOLD PTP P71 Vel=100 % PDAT51 Tool[1]:TOCH Base[0];%{PE}%R 8.3.48,%MKUKATPBASIS,%CMOVE,%VPTP,%P 1:PTP, 2:P71, 3:, 5:100, 7:PDAT51
$BWDSTART=FALSE
PDAT_ACT=PPDAT51
FDAT_ACT=FP71
BAS(#PTP_PARAMS,100)
PTP XP71
;ENDFOLD
;FOLD PTP P109 Vel=100 % PDAT85 Tool[1]:TOCH Base[0];%{PE}%R 8.3.48,%MKUKATPBASIS,%CMOVE,%VPTP,%P 1:PTP, 2:P109, 3:, 5:100, 7:PDAT85
$BWDSTART=FALSE
PDAT_ACT=PPDAT85
FDAT_ACT=FP109
BAS(#PTP_PARAMS,100)
PTP XP109
;ENDFOLD
;FOLD ; CORDAO 22;%{PE}%R 8.3.48,%MKUKATPBASIS,%CCOMMENT,%VNORMAL,%P 2:CORDAO 22
;ENDFOLD
;FOLD ARCON WDAT43 PTP P72 Vel=30 % PDAT52 Tool[1]:TOCH Base[0] ;%{PE}
;FOLD Parameters ;%{h}
;Params IlfProvider=kukaroboter.arctech.arconptp; Kuka.PointName=P72; Kuka.BlendingEnabled=False; Kuka.MoveDataPtpName=PDAT52; Kuka.VelocityPtp=30; Kuka.MovementParameterFieldEnabled=True; ArcTech.WdatVarName=WDAT43; ArcTech.SeamName=
;ENDFOLD
$BWDSTART = FALSE
PDAT_ACT = PPDAT52
FDAT_ACT = FP72
BAS(#PTP_PARAMS, 30.0)
TRIGGER WHEN DISTANCE = 1 DELAY = ATBg_PreDefinitionTime DO Arc_DefineStrikeParams(3, AS_WDAT43) PRIO = -1
Arc_DefineCpPattern(#OffInAdvance, WV_WDAT43, TRUE)
PTP XP72
Arc_On(1, AS_WDAT43, ATBg_StartErrSetField[1], AW_WDAT43, WV_WDAT43, ATBg_WeldErrSetField[1], #StdArcOn, " ")
Arc_DefineCpPattern(#OnInAdvance, WV_WDAT43, TRUE)
;ENDFOLD
;FOLD ARCOFF WDAT44 LIN P73 CPDAT23 Tool[1]:TOCH Base[0] ;%{PE}
;FOLD Parameters ;%{h}
;Params IlfProvider=kukaroboter.arctech.arcofflin; Kuka.PointName=P73; Kuka.BlendingEnabled=False; Kuka.MoveDataName=CPDAT23;  Kuka.MovementParameterFieldEnabled=True; ArcTech.WdatVarName=WDAT44
;ENDFOLD
$BWDSTART = FALSE
LDAT_ACT = LCPDAT23
FDAT_ACT = FP73
BAS(#CP_PARAMS, ATBg_BAS_VELDefinition)
LIN XP73
Arc_Off(1, AC_WDAT44)
;ENDFOLD
;FOLD PTP P74 Vel=100 % PDAT53 Tool[1]:TOCH Base[0];%{PE}%R 8.3.48,%MKUKATPBASIS,%CMOVE,%VPTP,%P 1:PTP, 2:P74, 3:, 5:100, 7:PDAT53
$BWDSTART=FALSE
PDAT_ACT=PPDAT53
FDAT_ACT=FP74
BAS(#PTP_PARAMS,100)
PTP XP74
;ENDFOLD
;FOLD PTP P103 Vel=100 % PDAT79 Tool[1]:TOCH Base[0];%{PE}%R 8.3.48,%MKUKATPBASIS,%CMOVE,%VPTP,%P 1:PTP, 2:P103, 3:, 5:100, 7:PDAT79
$BWDSTART=FALSE
PDAT_ACT=PPDAT79
FDAT_ACT=FP103
BAS(#PTP_PARAMS,100)
PTP XP103
;ENDFOLD
;FOLD ; CORDAO 23;%{PE}%R 8.3.48,%MKUKATPBASIS,%CCOMMENT,%VNORMAL,%P 2:CORDAO 23
;ENDFOLD
;FOLD ARCON WDAT45 PTP P75 Vel=30 % PDAT54 Tool[1]:TOCH Base[0] ;%{PE}
;FOLD Parameters ;%{h}
;Params IlfProvider=kukaroboter.arctech.arconptp; Kuka.PointName=P75; Kuka.BlendingEnabled=False; Kuka.MoveDataPtpName=PDAT54; Kuka.VelocityPtp=30; Kuka.MovementParameterFieldEnabled=True; ArcTech.WdatVarName=WDAT45; ArcTech.SeamName=
;ENDFOLD
$BWDSTART = FALSE
PDAT_ACT = PPDAT54
FDAT_ACT = FP75
BAS(#PTP_PARAMS, 30.0)
TRIGGER WHEN DISTANCE = 1 DELAY = ATBg_PreDefinitionTime DO Arc_DefineStrikeParams(3, AS_WDAT45) PRIO = -1
Arc_DefineCpPattern(#OffInAdvance, WV_WDAT45, TRUE)
PTP XP75
Arc_On(1, AS_WDAT45, ATBg_StartErrSetField[1], AW_WDAT45, WV_WDAT45, ATBg_WeldErrSetField[1], #StdArcOn, " ")
Arc_DefineCpPattern(#OnInAdvance, WV_WDAT45, TRUE)
;ENDFOLD
;FOLD ARCOFF WDAT46 LIN P76 CPDAT24 Tool[1]:TOCH Base[0] ;%{PE}
;FOLD Parameters ;%{h}
;Params IlfProvider=kukaroboter.arctech.arcofflin; Kuka.PointName=P76; Kuka.BlendingEnabled=False; Kuka.MoveDataName=CPDAT24;  Kuka.MovementParameterFieldEnabled=True; ArcTech.WdatVarName=WDAT46
;ENDFOLD
$BWDSTART = FALSE
LDAT_ACT = LCPDAT24
FDAT_ACT = FP76
BAS(#CP_PARAMS, ATBg_BAS_VELDefinition)
LIN XP76
Arc_Off(1, AC_WDAT46)
;ENDFOLD
;FOLD PTP P77 Vel=100 % PDAT55 Tool[1]:TOCH Base[0];%{PE}%R 8.3.48,%MKUKATPBASIS,%CMOVE,%VPTP,%P 1:PTP, 2:P77, 3:, 5:100, 7:PDAT55
$BWDSTART=FALSE
PDAT_ACT=PPDAT55
FDAT_ACT=FP77
BAS(#PTP_PARAMS,100)
PTP XP77
;ENDFOLD
;FOLD PTP P104 Vel=100 % PDAT80 Tool[1]:TOCH Base[0];%{PE}%R 8.3.48,%MKUKATPBASIS,%CMOVE,%VPTP,%P 1:PTP, 2:P104, 3:, 5:100, 7:PDAT80
$BWDSTART=FALSE
PDAT_ACT=PPDAT80
FDAT_ACT=FP104
BAS(#PTP_PARAMS,100)
PTP XP104
;ENDFOLD
;FOLD ; CORDAO 24;%{PE}%R 8.3.48,%MKUKATPBASIS,%CCOMMENT,%VNORMAL,%P 2:CORDAO 24
;ENDFOLD
;FOLD ARCON WDAT47 PTP P78 Vel=30 % PDAT56 Tool[1]:TOCH Base[0] ;%{PE}
;FOLD Parameters ;%{h}
;Params IlfProvider=kukaroboter.arctech.arconptp; Kuka.PointName=P78; Kuka.BlendingEnabled=False; Kuka.MoveDataPtpName=PDAT56; Kuka.VelocityPtp=30; Kuka.MovementParameterFieldEnabled=True; ArcTech.WdatVarName=WDAT47; ArcTech.SeamName=
;ENDFOLD
$BWDSTART = FALSE
PDAT_ACT = PPDAT56
FDAT_ACT = FP78
BAS(#PTP_PARAMS, 30.0)
TRIGGER WHEN DISTANCE = 1 DELAY = ATBg_PreDefinitionTime DO Arc_DefineStrikeParams(3, AS_WDAT47) PRIO = -1
Arc_DefineCpPattern(#OffInAdvance, WV_WDAT47, TRUE)
PTP XP78
Arc_On(1, AS_WDAT47, ATBg_StartErrSetField[1], AW_WDAT47, WV_WDAT47, ATBg_WeldErrSetField[1], #StdArcOn, " ")
Arc_DefineCpPattern(#OnInAdvance, WV_WDAT47, TRUE)
;ENDFOLD
;FOLD ARCOFF WDAT48 LIN P79 CPDAT25 Tool[1]:TOCH Base[0] ;%{PE}
;FOLD Parameters ;%{h}
;Params IlfProvider=kukaroboter.arctech.arcofflin; Kuka.PointName=P79; Kuka.BlendingEnabled=False; Kuka.MoveDataName=CPDAT25;  Kuka.MovementParameterFieldEnabled=True; ArcTech.WdatVarName=WDAT48
;ENDFOLD
$BWDSTART = FALSE
LDAT_ACT = LCPDAT25
FDAT_ACT = FP79
BAS(#CP_PARAMS, ATBg_BAS_VELDefinition)
LIN XP79
Arc_Off(1, AC_WDAT48)
;ENDFOLD
;FOLD PTP P105 Vel=100 % PDAT81 Tool[1]:TOCH Base[0];%{PE}%R 8.3.48,%MKUKATPBASIS,%CMOVE,%VPTP,%P 1:PTP, 2:P105, 3:, 5:100, 7:PDAT81
$BWDSTART=FALSE
PDAT_ACT=PPDAT81
FDAT_ACT=FP105
BAS(#PTP_PARAMS,100)
PTP XP105
;ENDFOLD
;FOLD PTP P80 Vel=100 % PDAT57 Tool[1]:TOCH Base[0];%{PE}%R 8.3.48,%MKUKATPBASIS,%CMOVE,%VPTP,%P 1:PTP, 2:P80, 3:, 5:100, 7:PDAT57
$BWDSTART=FALSE
PDAT_ACT=PPDAT57
FDAT_ACT=FP80
BAS(#PTP_PARAMS,100)
PTP XP80
;ENDFOLD
;FOLD ; CORDAO 24;%{PE}%R 8.3.48,%MKUKATPBASIS,%CCOMMENT,%VNORMAL,%P 2:CORDAO 24
;ENDFOLD
;FOLD ARCON WDAT49 PTP P81 Vel=30 % PDAT58 Tool[1]:TOCH Base[0] ;%{PE}
;FOLD Parameters ;%{h}
;Params IlfProvider=kukaroboter.arctech.arconptp; Kuka.PointName=P81; Kuka.BlendingEnabled=False; Kuka.MoveDataPtpName=PDAT58; Kuka.VelocityPtp=30; Kuka.MovementParameterFieldEnabled=True; ArcTech.WdatVarName=WDAT49; ArcTech.SeamName=
;ENDFOLD
$BWDSTART = FALSE
PDAT_ACT = PPDAT58
FDAT_ACT = FP81
BAS(#PTP_PARAMS, 30.0)
TRIGGER WHEN DISTANCE = 1 DELAY = ATBg_PreDefinitionTime DO Arc_DefineStrikeParams(3, AS_WDAT49) PRIO = -1
Arc_DefineCpPattern(#OffInAdvance, WV_WDAT49, TRUE)
PTP XP81
Arc_On(1, AS_WDAT49, ATBg_StartErrSetField[1], AW_WDAT49, WV_WDAT49, ATBg_WeldErrSetField[1], #StdArcOn, " ")
Arc_DefineCpPattern(#OnInAdvance, WV_WDAT49, TRUE)
;ENDFOLD
;FOLD ARCOFF WDAT50 LIN P82 CPDAT26 Tool[1]:TOCH Base[0] ;%{PE}
;FOLD Parameters ;%{h}
;Params IlfProvider=kukaroboter.arctech.arcofflin; Kuka.PointName=P82; Kuka.BlendingEnabled=False; Kuka.MoveDataName=CPDAT26;  Kuka.MovementParameterFieldEnabled=True; ArcTech.WdatVarName=WDAT50
;ENDFOLD
$BWDSTART = FALSE
LDAT_ACT = LCPDAT26
FDAT_ACT = FP82
BAS(#CP_PARAMS, ATBg_BAS_VELDefinition)
LIN XP82
Arc_Off(1, AC_WDAT50)
;ENDFOLD
;FOLD PTP P83 Vel=100 % PDAT59 Tool[1]:TOCH Base[0];%{PE}%R 8.3.48,%MKUKATPBASIS,%CMOVE,%VPTP,%P 1:PTP, 2:P83, 3:, 5:100, 7:PDAT59
$BWDSTART=FALSE
PDAT_ACT=PPDAT59
FDAT_ACT=FP83
BAS(#PTP_PARAMS,100)
PTP XP83
;ENDFOLD
;FOLD PTP P106 Vel=100 % PDAT82 Tool[1]:TOCH Base[0];%{PE}%R 8.3.48,%MKUKATPBASIS,%CMOVE,%VPTP,%P 1:PTP, 2:P106, 3:, 5:100, 7:PDAT82
$BWDSTART=FALSE
PDAT_ACT=PPDAT82
FDAT_ACT=FP106
BAS(#PTP_PARAMS,100)
PTP XP106
;ENDFOLD
;FOLD ; CORDAO 25;%{PE}%R 8.3.48,%MKUKATPBASIS,%CCOMMENT,%VNORMAL,%P 2:CORDAO 25
;ENDFOLD
;FOLD ARCON WDAT51 PTP P84 Vel=30 % PDAT60 Tool[1]:TOCH Base[0] ;%{PE}
;FOLD Parameters ;%{h}
;Params IlfProvider=kukaroboter.arctech.arconptp; Kuka.PointName=P84; Kuka.BlendingEnabled=False; Kuka.MoveDataPtpName=PDAT60; Kuka.VelocityPtp=30; Kuka.MovementParameterFieldEnabled=True; ArcTech.WdatVarName=WDAT51; ArcTech.SeamName=
;ENDFOLD
$BWDSTART = FALSE
PDAT_ACT = PPDAT60
FDAT_ACT = FP84
BAS(#PTP_PARAMS, 30.0)
TRIGGER WHEN DISTANCE = 1 DELAY = ATBg_PreDefinitionTime DO Arc_DefineStrikeParams(3, AS_WDAT51) PRIO = -1
Arc_DefineCpPattern(#OffInAdvance, WV_WDAT51, TRUE)
PTP XP84
Arc_On(1, AS_WDAT51, ATBg_StartErrSetField[1], AW_WDAT51, WV_WDAT51, ATBg_WeldErrSetField[1], #StdArcOn, " ")
Arc_DefineCpPattern(#OnInAdvance, WV_WDAT51, TRUE)
;ENDFOLD
;FOLD ARCOFF WDAT52 LIN P85 CPDAT27 Tool[1]:TOCH Base[0] ;%{PE}
;FOLD Parameters ;%{h}
;Params IlfProvider=kukaroboter.arctech.arcofflin; Kuka.PointName=P85; Kuka.BlendingEnabled=False; Kuka.MoveDataName=CPDAT27;  Kuka.MovementParameterFieldEnabled=True; ArcTech.WdatVarName=WDAT52
;ENDFOLD
$BWDSTART = FALSE
LDAT_ACT = LCPDAT27
FDAT_ACT = FP85
BAS(#CP_PARAMS, ATBg_BAS_VELDefinition)
LIN XP85
Arc_Off(1, AC_WDAT52)
;ENDFOLD
;FOLD PTP P86 Vel=100 % PDAT61 Tool[1]:TOCH Base[0];%{PE}%R 8.3.48,%MKUKATPBASIS,%CMOVE,%VPTP,%P 1:PTP, 2:P86, 3:, 5:100, 7:PDAT61
$BWDSTART=FALSE
PDAT_ACT=PPDAT61
FDAT_ACT=FP86
BAS(#PTP_PARAMS,100)
PTP XP86
;ENDFOLD
ENDLOOP
;FOLD PTP HOME Vel=100 % DEFAULT;%{PE}%R 8.3.48,%MKUKATPBASIS,%CMOVE,%VPTP,%P 1:PTP, 2:HOME, 3:, 5:100, 7:DEFAULT
$BWDSTART=FALSE
PDAT_ACT=PDEFAULT
FDAT_ACT=FHOME
BAS(#PTP_PARAMS,100)
$H_POS=XHOME
PTP XHOME
;ENDFOLD
END

--- MASTER_MESA_A.dat ---
&ACCESS RVP
&REL 294
&PARAM EDITMASK = *
&PARAM TEMPLATE = C:\KRC\Roboter\Template\vorgabe
&PARAM DISKPATH = KRC:\R1\Program\Solda
DEFDAT  MASTER_MESA_A
;FOLD EXTERNAL DECLARATIONS;%{PE}%MKUKATPBASIS,%CEXT,%VCOMMON,%P
;FOLD BASISTECH EXT;%{PE}%MKUKATPBASIS,%CEXT,%VEXT,%P
EXT  BAS (BAS_COMMAND  :IN,REAL  :IN )
DECL INT SUCCESS
;ENDFOLD (BASISTECH EXT)
;FOLD USER EXT;%{E}%MKUKATPUSER,%CEXT,%VEXT,%P
;Make your modifications here

;ENDFOLD (USER EXT)
;ENDFOLD (EXTERNAL DECLARATIONS)
DECL BASIS_SUGG_T LAST_BASIS={POINT1[] "P109                    ",POINT2[] "P109                    ",CP_PARAMS[] "CPDAT0                  ",PTP_PARAMS[] "PDAT85                  ",CONT[] "                        ",CP_VEL[] "2.0                     ",PTP_VEL[] "100                     ",SYNC_PARAMS[] "SYNCDAT                 ",SPL_NAME[] "S0                      ",A_PARAMS[] "ADAT0                   "}
DECL ATBg_Start_T AS_WDAT1={JobModeId 1306102413,ParamSetId -1047099609,StartTime 0.0,PreFlowTime 0.0,Channel1 0.0,Channel2 2.00000,Channel3 0.0,Channel4 0.0,Channel5 0.0,Channel6 0.0,Channel7 0.0,Channel8 0.0,PurgeTime 0.0}
DECL ATBg_Weld_T AW_WDAT1={JobModeId -187662529,ParamSetId -430485013,Velocity 0.00830000,Channel1 30.0000,Channel2 1.00000,Channel3 0.0,Channel4 0.0,Channel5 0.0,Channel6 0.0,Channel7 0.0,Channel8 0.0}
DECL WTCg_WeaveDefinition_T WV_WDAT1={Pattern #None,Length 4.00000,Amplitude 2.00000,Angle 0.0}
DECL FDAT FP1={TOOL_NO 1,BASE_NO 0,IPO_FRAME #BASE,POINT2[] " ",TQ_STATE FALSE}
DECL PDAT PPDAT1={ACC 100.000,APO_DIST 100.000,APO_MODE #CPTP,GEAR_JERK 50.0000}
DECL E6POS XP1={X 1366.71277,Y 550.959900,Z 1425.20300,A 20.2994423,B 41.1756821,C -155.754684,S 0,T 35,E1 193.394135,E2 193.959656,E3 193.454315,E4 0.0,E5 0.0,E6 0.0}
DECL MODULEPARAM_T LAST_TP_PARAMS={PARAMS[] "Kuka.MoveDataPtpName=PDAT60; Kuka.VelocityPtp=30; Kuka.PointName=P84; Kuka.BlendingEnabled=False; Kuka.FrameData.tq_state=False; Kuka.FrameData.base_no=0; Kuka.FrameData.tool_no=1; Kuka.FrameData.ipo_frame=#BASE; Kuka.MovementDataPdat.apo_mode=#CPTP; Kuka.MovementDataPdat.apo_dist=100; Kuka.MovementData.acc=100; Kuka.MovementData.gear_jerk=50; ArcTech.WdatVarName=WDAT51; Kuka.MoveDataName=CPDAT28; Kuka.VelocityPath=2; Kuka.FrameData.point2=; Kuka.MovementData.apo_fac=50; Kuka.MovementData.apo_dist=100; Kuka.MovementData.axis_acc=100; Kuka.MovementData.axis_vel=100; Kuka.MovementData.circ_typ=#BASE; Kuka.MovementData.exax_ign=0; Kuka.MovementData.jerk_fac=50; Kuka.MovementData.ori_typ=#VAR                                                                                                                                                                                                                           "}
DECL LDAT LCPDAT1={ACC 100.000,APO_DIST 100.000,APO_FAC 50.0000,AXIS_VEL 100.000,AXIS_ACC 100.000,ORI_TYP #VAR,CIRC_TYP #BASE,JERK_FAC 50.0000,GEAR_JERK 50.0000,EXAX_IGN 0}
DECL ATBg_Crater_T AC_WDAT2={JobModeId -187662529,ParamSetId -1375177600,CraterTime 0.100000,PostflowTime 0.100000,Channel1 30.0000,Channel2 1.00000,Channel3 0.0,Channel4 0.0,Channel5 0.0,Channel6 0.0,Channel7 0.0,Channel8 0.0,BurnBackTime 0.0}
DECL FDAT FP2={TOOL_NO 1,BASE_NO 0,IPO_FRAME #BASE,POINT2[] " ",TQ_STATE FALSE}
DECL LDAT LCPDAT2={ACC 100.000,APO_DIST 100.000,APO_FAC 50.0000,AXIS_VEL 100.000,AXIS_ACC 100.000,ORI_TYP #VAR,CIRC_TYP #BASE,JERK_FAC 50.0000,GEAR_JERK 50.0000,EXAX_IGN 0}
DECL E6POS XP2={X 1361.37756,Y 564.350647,Z 1425.89197,A 20.8604565,B 40.8836288,C -155.754288,S 0,T 35,E1 193.394135,E2 193.959656,E3 193.454315,E4 0.0,E5 0.0,E6 0.0}
DECL PDAT PPDAT2={ACC 100.000,APO_DIST 100.000,APO_MODE #CPTP,GEAR_JERK 50.0000}
DECL E6POS XP3={X 1149.30737,Y 478.114502,Z 1667.35852,A 20.0544758,B 29.3165226,C -165.776184,S 0,T 35,E1 193.394135,E2 193.959656,E3 193.454315,E4 0.0,E5 0.0,E6 0.0}
DECL FDAT FP3={TOOL_NO 1,BASE_NO 0,IPO_FRAME #BASE,POINT2[] " ",TQ_STATE FALSE}
DECL PDAT PPDAT3={VEL 100.000,ACC 100.000,APO_DIST 100.000,GEAR_JERK 50.0000,EXAX_IGN 3}
DECL E6POS XP4={X 1311.09155,Y 520.681274,Z 1579.92249,A 19.5462513,B 23.9474430,C -162.250244,S 2,T 35,E1 193.394135,E2 193.959656,E3 193.454315,E4 0.0,E5 0.0,E6 0.0}
DECL FDAT FP4={TOOL_NO 1,BASE_NO 0,IPO_FRAME #BASE,POINT2[] " ",TQ_STATE FALSE}
DECL PDAT PPDAT4={VEL 100.000,ACC 100.000,APO_DIST 100.000,GEAR_JERK 50.0000,EXAX_IGN 3}
DECL E6POS XP5={X 1311.09070,Y 575.770874,Z 1673.74915,A 27.2506332,B 22.9505119,C -67.7718811,S 2,T 35,E1 193.394135,E2 193.959656,E3 193.454315,E4 0.0,E5 0.0,E6 0.0}
DECL FDAT FP5={TOOL_NO 1,BASE_NO 0,IPO_FRAME #BASE,POINT2[] " ",TQ_STATE FALSE}
DECL PDAT PPDAT5={VEL 100.000,ACC 100.000,APO_DIST 100.000,GEAR_JERK 50.0000,EXAX_IGN 3}
DECL ATBg_Start_T AS_WDAT3={JobModeId 1306102413,ParamSetId -1047099609,StartTime 0.0,PreFlowTime 0.0,Channel1 0.0,Channel2 2.00000,Channel3 0.0,Channel4 0.0,Channel5 0.0,Channel6 0.0,Channel7 0.0,Channel8 0.0,PurgeTime 0.0}
DECL ATBg_Weld_T AW_WDAT3={JobModeId -187662529,ParamSetId -430485013,Velocity 0.00830000,Channel1 30.0000,Channel2 1.00000,Channel3 0.0,Channel4 0.0,Channel5 0.0,Channel6 0.0,Channel7 0.0,Channel8 0.0}
DECL WTCg_WeaveDefinition_T WV_WDAT3={Pattern #None,Length 4.00000,Amplitude 2.00000,Angle 0.0}
DECL FDAT FP6={TOOL_NO 1,BASE_NO 0,IPO_FRAME #BASE,POINT2[] " ",TQ_STATE FALSE}
DECL PDAT PPDAT6={ACC 100.000,APO_DIST 100.000,APO_MODE #CPTP,GEAR_JERK 50.0000}
DECL E6POS XP6={X 1335.21,Y 615.450745,Z 1642.98645,A 25.4925518,B 25.5691261,C -61.4651718,S 2,T 35,E1 193.394135,E2 193.959656,E3 193.454315,E4 0.0,E5 0.0,E6 0.0}
DECL ATBg_Crater_T AC_WDAT4={JobModeId -187662529,ParamSetId -1375177600,CraterTime 0.100000,PostflowTime 0.100000,Channel1 30.0000,Channel2 1.00000,Channel3 0.0,Channel4 0.0,Channel5 0.0,Channel6 0.0,Channel7 0.0,Channel8 0.0,BurnBackTime 0.0}
DECL FDAT FP7={TOOL_NO 1,BASE_NO 0,IPO_FRAME #BASE,POINT2[] " ",TQ_STATE FALSE}
DECL LDAT LCPDAT3={ACC 100.000,APO_DIST 100.000,APO_FAC 50.0000,AXIS_VEL 100.000,AXIS_ACC 100.000,ORI_TYP #VAR,CIRC_TYP #BASE,JERK_FAC 50.0000,GEAR_JERK 50.0000,EXAX_IGN 0}
DECL E6POS XP7={X 1324.19678,Y 623.090759,Z 1631.38159,A 25.8055401,B 27.3090305,C -67.4592743,S 2,T 35,E1 193.394135,E2 193.959656,E3 193.454315,E4 0.0,E5 0.0,E6 0.0}
DECL E6POS XP8={X 1279.20923,Y 604.527222,Z 1683.27698,A 25.7392673,B 25.0037098,C -67.6095810,S 2,T 35,E1 193.394135,E2 193.959656,E3 193.454315,E4 0.0,E5 0.0,E6 0.0}
DECL FDAT FP8={TOOL_NO 1,BASE_NO 0,IPO_FRAME #BASE,POINT2[] " ",TQ_STATE FALSE}
DECL PDAT PPDAT7={VEL 100.000,ACC 100.000,APO_DIST 100.000,GEAR_JERK 50.0000,EXAX_IGN 3}
DECL ATBg_Start_T AS_WDAT5={JobModeId 1306102413,ParamSetId -1047099609,StartTime 0.0,PreFlowTime 0.0,Channel1 0.0,Channel2 2.00000,Channel3 0.0,Channel4 0.0,Channel5 0.0,Channel6 0.0,Channel7 0.0,Channel8 0.0,PurgeTime 0.0}
DECL ATBg_Weld_T AW_WDAT5={JobModeId -187662529,ParamSetId -430485013,Velocity 0.00830000,Channel1 30.0000,Channel2 1.00000,Channel3 0.0,Channel4 0.0,Channel5 0.0,Channel6 0.0,Channel7 0.0,Channel8 0.0}
DECL WTCg_WeaveDefinition_T WV_WDAT5={Pattern #None,Length 4.00000,Amplitude 2.00000,Angle 0.0}
DECL FDAT FP9={TOOL_NO 1,BASE_NO 0,IPO_FRAME #BASE,POINT2[] " ",TQ_STATE FALSE}
DECL PDAT PPDAT8={ACC 100.000,APO_DIST 100.000,APO_MODE #CPTP,GEAR_JERK 50.0000}
DECL E6POS XP9={X 1338.59033,Y 603.315796,Z 1660.03796,A 23.5751057,B 18.2270985,C 28.4891853,S 2,T 35,E1 193.394135,E2 193.959656,E3 193.454315,E4 0.0,E5 0.0,E6 0.0}
DECL ATBg_Crater_T AC_WDAT6={JobModeId -187662529,ParamSetId -1375177600,CraterTime 0.100000,PostflowTime 0.100000,Channel1 30.0000,Channel2 1.00000,Channel3 0.0,Channel4 0.0,Channel5 0.0,Channel6 0.0,Channel7 0.0,Channel8 0.0,BurnBackTime 0.0}
DECL FDAT FP10={TOOL_NO 1,BASE_NO 0,IPO_FRAME #BASE,POINT2[] " ",TQ_STATE FALSE}
DECL LDAT LCPDAT4={ACC 100.000,APO_DIST 100.000,APO_FAC 50.0000,AXIS_VEL 100.000,AXIS_ACC 100.000,ORI_TYP #VAR,CIRC_TYP #BASE,JERK_FAC 50.0000,GEAR_JERK 50.0000,EXAX_IGN 0}
DECL E6POS XP10={X 1341.28662,Y 591.207458,Z 1658.64465,A 22.9818192,B 18.3544273,C 30.1838589,S 2,T 35,E1 193.394135,E2 193.959656,E3 193.454315,E4 0.0,E5 0.0,E6 0.0}
DECL E6POS XP11={X 928.621765,Y 202.400635,Z 1989.42310,A 17.9765,B 2.56140208,C 11.0882387,S 2,T 43,E1 193.394135,E2 193.959656,E3 193.454315,E4 0.0,E5 0.0,E6 0.0}
DECL FDAT FP11={TOOL_NO 1,BASE_NO 0,IPO_FRAME #BASE,POINT2[] " ",TQ_STATE FALSE}
DECL PDAT PPDAT9={VEL 100.000,ACC 100.000,APO_DIST 100.000,GEAR_JERK 50.0000,EXAX_IGN 3}
DECL E6POS XP12={X 1010.45526,Y 461.386902,Z 1947.43762,A 29.4855576,B 3.20235252,C 29.0299263,S 2,T 43,E1 193.394135,E2 193.959656,E3 193.454315,E4 0.0,E5 0.0,E6 0.0}
DECL FDAT FP12={TOOL_NO 1,BASE_NO 0,IPO_FRAME #BASE,POINT2[] " ",TQ_STATE FALSE}
DECL PDAT PPDAT10={VEL 100.000,ACC 100.000,APO_DIST 100.000,GEAR_JERK 50.0000,EXAX_IGN 3}
DECL E6POS XP13={X 1295.38977,Y 583.677368,Z 1687.53955,A 27.8626652,B 25.3438969,C 33.8667564,S 2,T 43,E1 193.394135,E2 193.959656,E3 193.454315,E4 0.0,E5 0.0,E6 0.0}
DECL FDAT FP13={TOOL_NO 1,BASE_NO 0,IPO_FRAME #BASE,POINT2[] " ",TQ_STATE FALSE}
DECL PDAT PPDAT11={VEL 100.000,ACC 100.000,APO_DIST 100.000,GEAR_JERK 50.0000,EXAX_IGN 3}
DECL ATBg_Start_T AS_WDAT7={JobModeId 1306102413,ParamSetId -1047099609,StartTime 0.0,PreFlowTime 0.0,Channel1 0.0,Channel2 2.00000,Channel3 0.0,Channel4 0.0,Channel5 0.0,Channel6 0.0,Channel7 0.0,Channel8 0.0,PurgeTime 0.0}
DECL ATBg_Weld_T AW_WDAT7={JobModeId -187662529,ParamSetId -430485013,Velocity 0.00830000,Channel1 30.0000,Channel2 1.00000,Channel3 0.0,Channel4 0.0,Channel5 0.0,Channel6 0.0,Channel7 0.0,Channel8 0.0}
DECL WTCg_WeaveDefinition_T WV_WDAT7={Pattern #None,Length 4.00000,Amplitude 2.00000,Angle 0.0}
DECL FDAT FP14={TOOL_NO 1,BASE_NO 0,IPO_FRAME #BASE,POINT2[] " ",TQ_STATE FALSE}
DECL PDAT PPDAT12={ACC 100.000,APO_DIST 100.000,APO_MODE #CPTP,GEAR_JERK 50.0000}
DECL E6POS XP14={X 1392.46790,Y 322.224060,Z 1673.09790,A 18.8083115,B 17.9801235,C 12.6240358,S 2,T 43,E1 193.394089,E2 193.959625,E3 193.454208,E4 0.0,E5 0.0,E6 0.0}
DECL ATBg_Crater_T AC_WDAT8={JobModeId -187662529,ParamSetId -1375177600,CraterTime 0.100000,PostflowTime 0.100000,Channel1 30.0000,Channel2 1.00000,Channel3 0.0,Channel4 0.0,Channel5 0.0,Channel6 0.0,Channel7 0.0,Channel8 0.0,BurnBackTime 0.0}
DECL FDAT FP15={TOOL_NO 1,BASE_NO 0,IPO_FRAME #BASE,POINT2[] " ",TQ_STATE FALSE}
DECL LDAT LCPDAT5={ACC 100.000,APO_DIST 100.000,APO_FAC 50.0000,AXIS_VEL 100.000,AXIS_ACC 100.000,ORI_TYP #VAR,CIRC_TYP #BASE,JERK_FAC 50.0000,GEAR_JERK 50.0000,EXAX_IGN 0}
DECL E6POS XP15={X 1396.25146,Y 303.561584,Z 1671.65527,A 18.0491753,B 18.1097832,C 12.6372776,S 2,T 43,E1 193.394089,E2 193.959625,E3 193.454208,E4 0.0,E5 0.0,E6 0.0}
DECL ATBg_Start_T AS_WDAT9={JobModeId 1306102413,ParamSetId -1047099609,StartTime 0.0,PreFlowTime 0.0,Channel1 0.0,Channel2 2.00000,Channel3 0.0,Channel4 0.0,Channel5 0.0,Channel6 0.0,Channel7 0.0,Channel8 0.0,PurgeTime 0.0}
DECL ATBg_Weld_T AW_WDAT9={JobModeId -187662529,ParamSetId -430485013,Velocity 0.00830000,Channel1 30.0000,Channel2 1.00000,Channel3 0.0,Channel4 0.0,Channel5 0.0,Channel6 0.0,Channel7 0.0,Channel8 0.0}
DECL WTCg_WeaveDefinition_T WV_WDAT9={Pattern #None,Length 4.00000,Amplitude 2.00000,Angle 0.0}
DECL FDAT FP16={TOOL_NO 1,BASE_NO 0,IPO_FRAME #BASE,POINT2[] " ",TQ_STATE FALSE}
DECL PDAT PPDAT13={ACC 100.000,APO_DIST 100.000,APO_MODE #CPTP,GEAR_JERK 50.0000}
DECL E6POS XP16={X 1409.85986,Y -21.9529438,Z 1672.00830,A 2.70648956,B 18.5833416,C 7.21969843,S 2,T 42,E1 193.394089,E2 193.959625,E3 193.454208,E4 0.0,E5 0.0,E6 0.0}
DECL ATBg_Crater_T AC_WDAT10={JobModeId -187662529,ParamSetId -1375177600,CraterTime 0.100000,PostflowTime 0.100000,Channel1 30.0000,Channel2 1.00000,Channel3 0.0,Channel4 0.0,Channel5 0.0,Channel6 0.0,Channel7 0.0,Channel8 0.0,BurnBackTime 0.0}
DECL FDAT FP17={TOOL_NO 1,BASE_NO 0,IPO_FRAME #BASE,POINT2[] " ",TQ_STATE FALSE}
DECL LDAT LCPDAT6={ACC 100.000,APO_DIST 100.000,APO_FAC 50.0000,AXIS_VEL 100.000,AXIS_ACC 100.000,ORI_TYP #VAR,CIRC_TYP #BASE,JERK_FAC 50.0000,GEAR_JERK 50.0000,EXAX_IGN 0}
DECL E6POS XP17={X 1409.10364,Y -3.69718385,Z 1673.18213,A 3.44733715,B 18.5231190,C 7.21611071,S 2,T 43,E1 193.394089,E2 193.959625,E3 193.454208,E4 0.0,E5 0.0,E6 0.0}
DECL E6POS XP18={X 1394.67908,Y -3.75147128,Z 1679.42834,A 3.44677186,B 18.4932098,C 7.21433,S 2,T 43,E1 193.394089,E2 193.959625,E3 193.454208,E4 0.0,E5 0.0,E6 0.0}
DECL FDAT FP18={TOOL_NO 1,BASE_NO 0,IPO_FRAME #BASE,POINT2[] " ",TQ_STATE FALSE}
DECL PDAT PPDAT14={VEL 100.000,ACC 100.000,APO_DIST 100.000,GEAR_JERK 50.0000,EXAX_IGN 3}
DECL E6POS XP19={X 1357.37805,Y 247.954,Z 1698.80786,A 15.7895479,B 17.5999718,C 11.7549076,S 2,T 43,E1 193.394089,E2 193.959625,E3 193.454208,E4 0.0,E5 0.0,E6 0.0}
DECL FDAT FP19={TOOL_NO 1,BASE_NO 0,IPO_FRAME #BASE,POINT2[] " ",TQ_STATE FALSE}
DECL PDAT PPDAT15={VEL 100.000,ACC 100.000,APO_DIST 100.000,GEAR_JERK 50.0000,EXAX_IGN 3}
DECL E6POS XP20={X 1360.18701,Y -3.88128376,Z 1710.14612,A 3.42260075,B 17.1567020,C 7.13537312,S 2,T 43,E1 193.394089,E2 193.959625,E3 193.454208,E4 0.0,E5 0.0,E6 0.0}
DECL FDAT FP20={TOOL_NO 1,BASE_NO 0,IPO_FRAME #BASE,POINT2[] " ",TQ_STATE FALSE}
DECL PDAT PPDAT16={VEL 100.000,ACC 100.000,APO_DIST 100.000,GEAR_JERK 50.0000,EXAX_IGN 3}
DECL E6POS XP21={X 1415.86548,Y -37.9887619,Z 1525.39063,A -3.52772069,B 31.1256237,C 173.144684,S 2,T 10,E1 193.394089,E2 193.959625,E3 193.454208,E4 0.0,E5 0.0,E6 0.0}
DECL FDAT FP21={TOOL_NO 1,BASE_NO 0,IPO_FRAME #BASE,POINT2[] " ",TQ_STATE FALSE}
DECL PDAT PPDAT17={VEL 100.000,ACC 100.000,APO_DIST 100.000,GEAR_JERK 50.0000,EXAX_IGN 3}
DECL ATBg_Start_T AS_WDAT11={JobModeId 1306102413,ParamSetId -1047099609,StartTime 0.0,PreFlowTime 0.0,Channel1 0.0,Channel2 2.00000,Channel3 0.0,Channel4 0.0,Channel5 0.0,Channel6 0.0,Channel7 0.0,Channel8 0.0,PurgeTime 0.0}
DECL ATBg_Weld_T AW_WDAT11={JobModeId -187662529,ParamSetId -430485013,Velocity 0.00830000,Channel1 30.0000,Channel2 1.00000,Channel3 0.0,Channel4 0.0,Channel5 0.0,Channel6 0.0,Channel7 0.0,Channel8 0.0}
DECL WTCg_WeaveDefinition_T WV_WDAT11={Pattern #None,Length 4.00000,Amplitude 2.00000,Angle 0.0}
DECL FDAT FP22={TOOL_NO 1,BASE_NO 0,IPO_FRAME #BASE,POINT2[] " ",TQ_STATE FALSE}
DECL PDAT PPDAT18={ACC 100.000,APO_DIST 100.000,APO_MODE #CPTP,GEAR_JERK 50.0000}
DECL E6POS XP22={X 1458.39331,Y -39.1287231,Z 1453.48657,A -3.65856624,B 36.4265099,C 172.919220,S 2,T 10,E1 193.394089,E2 193.959625,E3 193.454208,E4 0.0,E5 0.0,E6 0.0}
DECL ATBg_Crater_T AC_WDAT12={JobModeId -187662529,ParamSetId -1375177600,CraterTime 0.100000,PostflowTime 0.100000,Channel1 30.0000,Channel2 1.00000,Channel3 0.0,Channel4 0.0,Channel5 0.0,Channel6 0.0,Channel7 0.0,Channel8 0.0,BurnBackTime 0.0}
DECL FDAT FP23={TOOL_NO 1,BASE_NO 0,IPO_FRAME #BASE,POINT2[] " ",TQ_STATE FALSE}
DECL LDAT LCPDAT7={ACC 100.000,APO_DIST 100.000,APO_FAC 50.0000,AXIS_VEL 100.000,AXIS_ACC 100.000,ORI_TYP #VAR,CIRC_TYP #BASE,JERK_FAC 50.0000,GEAR_JERK 50.0000,EXAX_IGN 0}
DECL E6POS XP23={X 1458.80884,Y -17.8529091,Z 1453.48657,A -2.82283902,B 36.4265099,C 172.919220,S 2,T 10,E1 193.394089,E2 193.959625,E3 193.454208,E4 0.0,E5 0.0,E6 0.0}
DECL ATBg_Start_T AS_WDAT13={JobModeId 1306102413,ParamSetId -1047099609,StartTime 0.0,PreFlowTime 0.0,Channel1 0.0,Channel2 2.00000,Channel3 0.0,Channel4 0.0,Channel5 0.0,Channel6 0.0,Channel7 0.0,Channel8 0.0,PurgeTime 0.0}
DECL ATBg_Weld_T AW_WDAT13={JobModeId -187662529,ParamSetId -430485013,Velocity 0.00830000,Channel1 30.0000,Channel2 1.00000,Channel3 0.0,Channel4 0.0,Channel5 0.0,Channel6 0.0,Channel7 0.0,Channel8 0.0}
DECL WTCg_WeaveDefinition_T WV_WDAT13={Pattern #None,Length 4.00000,Amplitude 2.00000,Angle 0.0}
DECL FDAT FP24={TOOL_NO 1,BASE_NO 0,IPO_FRAME #BASE,POINT2[] " ",TQ_STATE FALSE}
DECL PDAT PPDAT19={ACC 100.000,APO_DIST 100.000,APO_MODE #CPTP,GEAR_JERK 50.0000}
DECL E6POS XP24={X 1427.31030,Y 336.997253,Z 1465.61572,A 12.9234352,B 36.0036659,C -158.134964,S 2,T 43,E1 193.394043,E2 193.959610,E3 193.454132,E4 0.0,E5 0.0,E6 0.0}
DECL ATBg_Crater_T AC_WDAT14={JobModeId -187662529,ParamSetId -1375177600,CraterTime 0.100000,PostflowTime 0.100000,Channel1 30.0000,Channel2 1.00000,Channel3 0.0,Channel4 0.0,Channel5 0.0,Channel6 0.0,Channel7 0.0,Channel8 0.0,BurnBackTime 0.0}
DECL FDAT FP25={TOOL_NO 1,BASE_NO 0,IPO_FRAME #BASE,POINT2[] " ",TQ_STATE FALSE}
DECL LDAT LCPDAT8={ACC 100.000,APO_DIST 100.000,APO_FAC 50.0000,AXIS_VEL 100.000,AXIS_ACC 100.000,ORI_TYP #VAR,CIRC_TYP #BASE,JERK_FAC 50.0000,GEAR_JERK 50.0000,EXAX_IGN 0}
DECL E6POS XP25={X 1430.67944,Y 319.374664,Z 1465.13574,A 12.2247372,B 36.1712227,C -158.130432,S 2,T 43,E1 193.394043,E2 193.959610,E3 193.454132,E4 0.0,E5 0.0,E6 0.0}
DECL E6POS XP26={X 1413.45007,Y 316.034943,Z 1492.89551,A 12.1964798,B 34.3249092,C -158.179382,S 2,T 43,E1 193.394043,E2 193.959610,E3 193.454132,E4 0.0,E5 0.0,E6 0.0}
DECL FDAT FP26={TOOL_NO 1,BASE_NO 0,IPO_FRAME #BASE,POINT2[] " ",TQ_STATE FALSE}
DECL PDAT PPDAT20={VEL 100.000,ACC 100.000,APO_DIST 100.000,GEAR_JERK 50.0000,EXAX_IGN 3}
DECL E6POS XP27={X 1413.45007,Y 316.034943,Z 1492.89551,A 12.1964798,B 34.3249092,C -158.179382,S 2,T 43,E1 193.394043,E2 193.959610,E3 193.454132,E4 0.0,E5 0.0,E6 0.0}
DECL FDAT FP27={TOOL_NO 1,BASE_NO 0,IPO_FRAME #BASE,POINT2[] " ",TQ_STATE FALSE}
DECL PDAT PPDAT21={VEL 100.000,ACC 100.000,APO_DIST 100.000,GEAR_JERK 50.0000,EXAX_IGN 3}
DECL E6POS XP28={X 1444.15625,Y -4.81991434,Z 1485.19397,A -1.90741491,B 34.0847778,C -177.298203,S 2,T 42,E1 193.394043,E2 193.959610,E3 193.454132,E4 0.0,E5 0.0,E6 0.0}
DECL FDAT FP28={TOOL_NO 1,BASE_NO 0,IPO_FRAME #BASE,POINT2[] " ",TQ_STATE FALSE}
DECL PDAT PPDAT22={VEL 100.000,ACC 100.000,APO_DIST 100.000,GEAR_JERK 50.0000,EXAX_IGN 3}
DECL ATBg_Start_T AS_WDAT15={JobModeId 1306102413,ParamSetId -1047099609,StartTime 0.0,PreFlowTime 0.0,Channel1 0.0,Channel2 2.00000,Channel3 0.0,Channel4 0.0,Channel5 0.0,Channel6 0.0,Channel7 0.0,Channel8 0.0,PurgeTime 0.0}
DECL ATBg_Weld_T AW_WDAT15={JobModeId -187662529,ParamSetId -430485013,Velocity 0.00830000,Channel1 30.0000,Channel2 1.00000,Channel3 0.0,Channel4 0.0,Channel5 0.0,Channel6 0.0,Channel7 0.0,Channel8 0.0}
DECL WTCg_WeaveDefinition_T WV_WDAT15={Pattern #None,Length 4.00000,Amplitude 2.00000,Angle 0.0}
DECL FDAT FP29={TOOL_NO 1,BASE_NO 0,IPO_FRAME #BASE,POINT2[] " ",TQ_STATE FALSE}
DECL PDAT PPDAT23={ACC 100.000,APO_DIST 100.000,APO_MODE #CPTP,GEAR_JERK 50.0000}
DECL E6POS XP29={X 1374.57507,Y -534.963440,Z 1471.28247,A -24.4083099,B 31.3126106,C 152.593872,S 0,T 10,E1 193.394,E2 193.959457,E3 193.454041,E4 0.0,E5 0.0,E6 0.0}
DECL ATBg_Crater_T AC_WDAT16={JobModeId -187662529,ParamSetId -1375177600,CraterTime 0.100000,PostflowTime 0.100000,Channel1 30.0000,Channel2 1.00000,Channel3 0.0,Channel4 0.0,Channel5 0.0,Channel6 0.0,Channel7 0.0,Channel8 0.0,BurnBackTime 0.0}
DECL FDAT FP30={TOOL_NO 1,BASE_NO 0,IPO_FRAME #BASE,POINT2[] " ",TQ_STATE FALSE}
DECL LDAT LCPDAT9={ACC 100.000,APO_DIST 100.000,APO_FAC 50.0000,AXIS_VEL 100.000,AXIS_ACC 100.000,ORI_TYP #VAR,CIRC_TYP #BASE,JERK_FAC 50.0000,GEAR_JERK 50.0000,EXAX_IGN 0}
DECL E6POS XP30={X 1371.93762,Y -546.517212,Z 1470.45776,A -24.8596382,B 31.1475182,C 152.612,S 0,T 10,E1 193.394,E2 193.959457,E3 193.454041,E4 0.0,E5 0.0,E6 0.0}
DECL E6POS XP31={X 1345.02637,Y -536.452576,Z 1514.93787,A -24.7163010,B 27.7588806,C 152.903381,S 0,T 10,E1 193.394,E2 193.959457,E3 193.454041,E4 0.0,E5 0.0,E6 0.0}
DECL FDAT FP31={TOOL_NO 1,BASE_NO 0,IPO_FRAME #BASE,POINT2[] " ",TQ_STATE FALSE}
DECL PDAT PPDAT24={VEL 100.000,ACC 100.000,APO_DIST 100.000,GEAR_JERK 50.0000,EXAX_IGN 3}
DECL E6POS XP32={X 1428.06470,Y -59.7406273,Z 1552.89087,A -4.16062450,B 24.3402233,C -177.736954,S 2,T 42,E1 193.394028,E2 193.959549,E3 193.454102,E4 0.0,E5 0.0,E6 0.0}
DECL FDAT FP32={TOOL_NO 1,BASE_NO 0,IPO_FRAME #BASE,POINT2[] " ",TQ_STATE FALSE}
DECL PDAT PPDAT25={VEL 100.000,ACC 100.000,APO_DIST 100.000,GEAR_JERK 50.0000,EXAX_IGN 3}
DECL E6POS XP33={X 1413.54114,Y -222.052826,Z 1555.41357,A -11.5825768,B 23.1373062,C 161.065216,S 2,T 10,E1 193.394028,E2 193.959549,E3 193.454102,E4 0.0,E5 0.0,E6 0.0}
DECL FDAT FP33={TOOL_NO 1,BASE_NO 0,IPO_FRAME #BASE,POINT2[] " ",TQ_STATE FALSE}
DECL PDAT PPDAT26={VEL 100.000,ACC 100.000,APO_DIST 100.000,GEAR_JERK 50.0000,EXAX_IGN 3}
DECL E6POS XP34={X 1359.79089,Y -485.537628,Z 1580.67517,A -22.2542496,B 16.2812424,C 161.599228,S 2,T 10,E1 193.394028,E2 193.959549,E3 193.454102,E4 0.0,E5 0.0,E6 0.0}
DECL FDAT FP34={TOOL_NO 1,BASE_NO 0,IPO_FRAME #BASE,POINT2[] " ",TQ_STATE FALSE}
DECL PDAT PPDAT27={VEL 100.000,ACC 100.000,APO_DIST 100.000,GEAR_JERK 50.0000,EXAX_IGN 3}
DECL ATBg_Start_T AS_WDAT17={JobModeId 1306102413,ParamSetId -1047099609,StartTime 0.0,PreFlowTime 0.0,Channel1 0.0,Channel2 2.00000,Channel3 0.0,Channel4 0.0,Channel5 0.0,Channel6 0.0,Channel7 0.0,Channel8 0.0,PurgeTime 0.0}
DECL ATBg_Weld_T AW_WDAT17={JobModeId -187662529,ParamSetId -430485013,Velocity 0.00830000,Channel1 30.0000,Channel2 1.00000,Channel3 0.0,Channel4 0.0,Channel5 0.0,Channel6 0.0,Channel7 0.0,Channel8 0.0}
DECL WTCg_WeaveDefinition_T WV_WDAT17={Pattern #None,Length 4.00000,Amplitude 2.00000,Angle 0.0}
DECL FDAT FP35={TOOL_NO 1,BASE_NO 0,IPO_FRAME #BASE,POINT2[] " ",TQ_STATE FALSE}
DECL PDAT PPDAT28={ACC 100.000,APO_DIST 100.000,APO_MODE #CPTP,GEAR_JERK 50.0000}
DECL E6POS XP35={X 1370.58740,Y -528.344299,Z 1644.78894,A -21.3700218,B 26.9062672,C -26.2295723,S 2,T 34,E1 193.394,E2 193.959457,E3 193.454041,E4 0.0,E5 0.0,E6 0.0}
DECL ATBg_Crater_T AC_WDAT18={JobModeId -187662529,ParamSetId -1375177600,CraterTime 0.100000,PostflowTime 0.100000,Channel1 30.0000,Channel2 1.00000,Channel3 0.0,Channel4 0.0,Channel5 0.0,Channel6 0.0,Channel7 0.0,Channel8 0.0,BurnBackTime 0.0}
DECL FDAT FP36={TOOL_NO 1,BASE_NO 0,IPO_FRAME #BASE,POINT2[] " ",TQ_STATE FALSE}
DECL LDAT LCPDAT10={ACC 100.000,APO_DIST 100.000,APO_FAC 50.0000,AXIS_VEL 100.000,AXIS_ACC 100.000,ORI_TYP #VAR,CIRC_TYP #BASE,JERK_FAC 50.0000,GEAR_JERK 50.0000,EXAX_IGN 0}
DECL E6POS XP36={X 1373.73499,Y -515.872742,Z 1643.23254,A -20.7828598,B 27.0032749,C -28.9675655,S 2,T 34,E1 193.394,E2 193.959457,E3 193.454041,E4 0.0,E5 0.0,E6 0.0}
DECL E6POS XP37={X 1265.18945,Y -582.384949,Z 1704.90552,A -24.9814968,B 25.0390682,C -28.9961643,S 2,T 34,E1 193.394,E2 193.959457,E3 193.454041,E4 0.0,E5 0.0,E6 0.0}
DECL FDAT FP37={TOOL_NO 1,BASE_NO 0,IPO_FRAME #BASE,POINT2[] " ",TQ_STATE FALSE}
DECL PDAT PPDAT29={VEL 100.000,ACC 100.000,APO_DIST 100.000,GEAR_JERK 50.0000,EXAX_IGN 3}
DECL E6POS XP38={X 1355.19800,Y -506.540283,Z 1658.14575,A -20.6953545,B 26.7519760,C -29.2852974,S 2,T 34,E1 193.394,E2 193.959457,E3 193.454041,E4 0.0,E5 0.0,E6 0.0}
DECL FDAT FP38={TOOL_NO 1,BASE_NO 0,IPO_FRAME #BASE,POINT2[] " ",TQ_STATE FALSE}
DECL PDAT PPDAT30={VEL 100.000,ACC 100.000,APO_DIST 100.000,GEAR_JERK 50.0000,EXAX_IGN 3}
DECL E6POS XP39={X 1190.28735,Y -487.713867,Z 1755.25635,A -25.0673046,B -16.7617149,C -179.491501,S 2,T 42,E1 193.394,E2 193.959457,E3 193.454041,E4 0.0,E5 0.0,E6 0.0}
DECL FDAT FP39={TOOL_NO 1,BASE_NO 0,IPO_FRAME #BASE,POINT2[] " ",TQ_STATE FALSE}
DECL PDAT PPDAT31={VEL 100.000,ACC 100.000,APO_DIST 100.000,GEAR_JERK 50.0000,EXAX_IGN 3}
DECL E6POS XP40={X 1222.53,Y -517.756958,Z 1705.24719,A -23.3703079,B -0.0642994121,C -134.348877,S 2,T 34,E1 193.394,E2 193.959457,E3 193.454041,E4 0.0,E5 0.0,E6 0.0}
DECL FDAT FP40={TOOL_NO 1,BASE_NO 0,IPO_FRAME #BASE,POINT2[] " ",TQ_STATE FALSE}
DECL PDAT PPDAT32={VEL 100.000,ACC 100.000,APO_DIST 100.000,GEAR_JERK 50.0000,EXAX_IGN 3}
DECL ATBg_Start_T AS_WDAT19={JobModeId 1306102413,ParamSetId -1047099609,StartTime 0.0,PreFlowTime 0.0,Channel1 0.0,Channel2 2.00000,Channel3 0.0,Channel4 0.0,Channel5 0.0,Channel6 0.0,Channel7 0.0,Channel8 0.0,PurgeTime 0.0}
DECL ATBg_Weld_T AW_WDAT19={JobModeId -187662529,ParamSetId -430485013,Velocity 0.00830000,Channel1 30.0000,Channel2 1.00000,Channel3 0.0,Channel4 0.0,Channel5 0.0,Channel6 0.0,Channel7 0.0,Channel8 0.0}
DECL WTCg_WeaveDefinition_T WV_WDAT19={Pattern #None,Length 4.00000,Amplitude 2.00000,Angle 0.0}
DECL FDAT FP41={TOOL_NO 1,BASE_NO 0,IPO_FRAME #BASE,POINT2[] " ",TQ_STATE FALSE}
DECL PDAT PPDAT33={ACC 100.000,APO_DIST 100.000,APO_MODE #CPTP,GEAR_JERK 50.0000}
DECL E6POS XP41={X 1327.79980,Y -560.767639,Z 1594.29456,A 1.08999431,B -5.53085136,C 155.584366,S 2,T 10,E1 193.394,E2 193.959457,E3 193.454041,E4 0.0,E5 0.0,E6 0.0}
DECL ATBg_Crater_T AC_WDAT20={JobModeId -187662529,ParamSetId -1375177600,CraterTime 0.100000,PostflowTime 0.100000,Channel1 30.0000,Channel2 1.00000,Channel3 0.0,Channel4 0.0,Channel5 0.0,Channel6 0.0,Channel7 0.0,Channel8 0.0,BurnBackTime 0.0}
DECL FDAT FP42={TOOL_NO 1,BASE_NO 0,IPO_FRAME #BASE,POINT2[] " ",TQ_STATE FALSE}
DECL LDAT LCPDAT11={ACC 100.000,APO_DIST 100.000,APO_FAC 50.0000,AXIS_VEL 100.000,AXIS_ACC 100.000,ORI_TYP #VAR,CIRC_TYP #BASE,JERK_FAC 50.0000,GEAR_JERK 50.0000,EXAX_IGN 0}
DECL E6POS XP42={X 1325.24902,Y -567.523743,Z 1597.78955,A -0.143767759,B -6.26507282,C 154.822159,S 2,T 10,E1 193.394,E2 193.959457,E3 193.454041,E4 0.0,E5 0.0,E6 0.0}
DECL ATBg_Start_T AS_WDAT21={JobModeId 1306102413,ParamSetId -1047099609,StartTime 0.0,PreFlowTime 0.0,Channel1 0.0,Channel2 2.00000,Channel3 0.0,Channel4 0.0,Channel5 0.0,Channel6 0.0,Channel7 0.0,Channel8 0.0,PurgeTime 0.0}
DECL ATBg_Weld_T AW_WDAT21={JobModeId -187662529,ParamSetId -430485013,Velocity 0.00830000,Channel1 30.0000,Channel2 1.00000,Channel3 0.0,Channel4 0.0,Channel5 0.0,Channel6 0.0,Channel7 0.0,Channel8 0.0}
DECL WTCg_WeaveDefinition_T WV_WDAT21={Pattern #None,Length 4.00000,Amplitude 2.00000,Angle 0.0}
DECL FDAT FP43={TOOL_NO 1,BASE_NO 0,IPO_FRAME #BASE,POINT2[] " ",TQ_STATE FALSE}
DECL PDAT PPDAT34={ACC 100.000,APO_DIST 100.000,APO_MODE #CPTP,GEAR_JERK 50.0000}
DECL E6POS XP43={X 1277.69800,Y -724.347168,Z 1635.13452,A -9.24587631,B -11.2834444,C 127.346405,S 2,T 10,E1 193.394,E2 193.959457,E3 193.454041,E4 0.0,E5 0.0,E6 0.0}
DECL ATBg_Crater_T AC_WDAT22={JobModeId -187662529,ParamSetId -1375177600,CraterTime 0.100000,PostflowTime 0.100000,Channel1 30.0000,Channel2 1.00000,Channel3 0.0,Channel4 0.0,Channel5 0.0,Channel6 0.0,Channel7 0.0,Channel8 0.0,BurnBackTime 0.0}
DECL FDAT FP44={TOOL_NO 1,BASE_NO 0,IPO_FRAME #BASE,POINT2[] " ",TQ_STATE FALSE}
DECL LDAT LCPDAT12={ACC 100.000,APO_DIST 100.000,APO_FAC 50.0000,AXIS_VEL 100.000,AXIS_ACC 100.000,ORI_TYP #VAR,CIRC_TYP #BASE,JERK_FAC 50.0000,GEAR_JERK 50.0000,EXAX_IGN 0}
DECL E6POS XP44={X 1277.69800,Y -724.347168,Z 1635.13452,A -9.24587631,B -11.2834444,C 127.346405,S 2,T 10,E1 193.394,E2 193.959457,E3 193.454041,E4 0.0,E5 0.0,E6 0.0}
DECL ATBg_Start_T AS_WDAT23={JobModeId -187662529,ParamSetId 687014726,StartTime 0.0,PreFlowTime 0.100000,Channel1 30.0000,Channel2 1.00000,Channel3 0.0,Channel4 0.0,Channel5 0.0,Channel6 0.0,Channel7 0.0,Channel8 0.0,PurgeTime 0.0}
DECL ATBg_Weld_T AW_WDAT23={JobModeId -187662529,ParamSetId -430485013,Velocity 0.00830000,Channel1 30.0000,Channel2 1.00000,Channel3 0.0,Channel4 0.0,Channel5 0.0,Channel6 0.0,Channel7 0.0,Channel8 0.0}
DECL WTCg_WeaveDefinition_T WV_WDAT23={Pattern #None,Length 4.00000,Amplitude 2.00000,Angle 0.0}
DECL FDAT FP45={TOOL_NO 1,BASE_NO 0,IPO_FRAME #BASE,POINT2[] " ",TQ_STATE FALSE}
DECL PDAT PPDAT35={ACC 100.000,APO_DIST 100.000,APO_MODE #CPTP,GEAR_JERK 50.0000}
DECL E6POS XP45={X 1285.36877,Y -701.800232,Z 1621.29614,A -7.54951525,B -9.75901794,C 138.375687,S 2,T 10,E1 193.394,E2 193.959457,E3 193.454041,E4 0.0,E5 0.0,E6 0.0}
DECL ATBg_Crater_T AC_WDAT24={JobModeId -187662529,ParamSetId -1375177600,CraterTime 0.100000,PostflowTime 0.100000,Channel1 30.0000,Channel2 1.00000,Channel3 0.0,Channel4 0.0,Channel5 0.0,Channel6 0.0,Channel7 0.0,Channel8 0.0,BurnBackTime 0.0}
DECL FDAT FP46={TOOL_NO 1,BASE_NO 0,IPO_FRAME #BASE,POINT2[] " ",TQ_STATE FALSE}
DECL LDAT LCPDAT13={ACC 100.000,APO_DIST 100.000,APO_FAC 50.0000,AXIS_VEL 100.000,AXIS_ACC 100.000,ORI_TYP #VAR,CIRC_TYP #BASE,JERK_FAC 50.0000,GEAR_JERK 50.0000,EXAX_IGN 0}
DECL E6POS XP46={X 1286.50220,Y -693.705505,Z 1623.65881,A -7.24915314,B -9.82592,C 138.346390,S 2,T 10,E1 193.394,E2 193.959457,E3 193.454041,E4 0.0,E5 0.0,E6 0.0}
DECL E6POS XP47={X 1269.99438,Y -673.679077,Z 1650.53772,A -6.85948944,B -11.0520535,C 133.720520,S 2,T 10,E1 193.394,E2 193.959457,E3 193.454041,E4 0.0,E5 0.0,E6 0.0}
DECL FDAT FP47={TOOL_NO 1,BASE_NO 0,IPO_FRAME #BASE,POINT2[] " ",TQ_STATE FALSE}
DECL PDAT PPDAT36={VEL 100.000,ACC 100.000,APO_DIST 100.000,GEAR_JERK 50.0000,EXAX_IGN 3}
DECL E6POS XP48={X 905.718445,Y -468.565399,Z 1971.60498,A -4.82598686,B -26.0840855,C 130.575607,S 2,T 10,E1 193.394,E2 193.959457,E3 193.454041,E4 0.0,E5 0.0,E6 0.0}
DECL FDAT FP48={TOOL_NO 1,BASE_NO 0,IPO_FRAME #BASE,POINT2[] " ",TQ_STATE FALSE}
DECL PDAT PPDAT37={VEL 100.000,ACC 100.000,APO_DIST 100.000,GEAR_JERK 50.0000,EXAX_IGN 3}
DECL ATBg_Start_T AS_WDAT25={JobModeId 1306102413,ParamSetId -1047099609,StartTime 0.0,PreFlowTime 0.0,Channel1 0.0,Channel2 2.00000,Channel3 0.0,Channel4 0.0,Channel5 0.0,Channel6 0.0,Channel7 0.0,Channel8 0.0,PurgeTime 0.0}
DECL ATBg_Weld_T AW_WDAT25={JobModeId -187662529,ParamSetId -430485013,Velocity 0.00830000,Channel1 30.0000,Channel2 1.00000,Channel3 0.0,Channel4 0.0,Channel5 0.0,Channel6 0.0,Channel7 0.0,Channel8 0.0}
DECL WTCg_WeaveDefinition_T WV_WDAT25={Pattern #None,Length 4.00000,Amplitude 2.00000,Angle 0.0}
DECL FDAT FP49={TOOL_NO 1,BASE_NO 0,IPO_FRAME #BASE,POINT2[] " ",TQ_STATE FALSE}
DECL PDAT PPDAT38={ACC 100.000,APO_DIST 100.000,APO_MODE #CPTP,GEAR_JERK 50.0000}
DECL E6POS XP49={X 1251.05591,Y -807.726501,Z 1598.14941,A -9.59379292,B -8.40495586,C 160.356506,S 2,T 10,E1 193.394,E2 193.959457,E3 193.454041,E4 0.0,E5 0.0,E6 0.0}
DECL ATBg_Crater_T AC_WDAT26={JobModeId -187662529,ParamSetId -1375177600,CraterTime 0.100000,PostflowTime 0.100000,Channel1 30.0000,Channel2 1.00000,Channel3 0.0,Channel4 0.0,Channel5 0.0,Channel6 0.0,Channel7 0.0,Channel8 0.0,BurnBackTime 0.0}
DECL FDAT FP50={TOOL_NO 1,BASE_NO 0,IPO_FRAME #BASE,POINT2[] " ",TQ_STATE FALSE}
DECL LDAT LCPDAT14={ACC 100.000,APO_DIST 100.000,APO_FAC 50.0000,AXIS_VEL 100.000,AXIS_ACC 100.000,ORI_TYP #VAR,CIRC_TYP #BASE,JERK_FAC 50.0000,GEAR_JERK 50.0000,EXAX_IGN 0}
DECL E6POS XP50={X 1249.71765,Y -816.140320,Z 1597.00928,A -9.87893295,B -8.48013878,C 160.317978,S 2,T 10,E1 193.394,E2 193.959457,E3 193.454041,E4 0.0,E5 0.0,E6 0.0}
DECL ATBg_Start_T AS_WDAT27={JobModeId 1306102413,ParamSetId -1047099609,StartTime 0.0,PreFlowTime 0.0,Channel1 0.0,Channel2 2.00000,Channel3 0.0,Channel4 0.0,Channel5 0.0,Channel6 0.0,Channel7 0.0,Channel8 0.0,PurgeTime 0.0}
DECL ATBg_Weld_T AW_WDAT27={JobModeId -187662529,ParamSetId -430485013,Velocity 0.00830000,Channel1 30.0000,Channel2 1.00000,Channel3 0.0,Channel4 0.0,Channel5 0.0,Channel6 0.0,Channel7 0.0,Channel8 0.0}
DECL WTCg_WeaveDefinition_T WV_WDAT27={Pattern #None,Length 4.00000,Amplitude 2.00000,Angle 0.0}
DECL FDAT FP51={TOOL_NO 1,BASE_NO 0,IPO_FRAME #BASE,POINT2[] " ",TQ_STATE FALSE}
DECL PDAT PPDAT39={ACC 100.000,APO_DIST 100.000,APO_MODE #CPTP,GEAR_JERK 50.0000}
DECL E6POS XP51={X 1242.06677,Y -827.762268,Z 1624.22620,A -10.8560162,B -10.8155499,C 136.973816,S 2,T 10,E1 193.394,E2 193.959457,E3 193.454041,E4 0.0,E5 0.0,E6 0.0}
DECL ATBg_Crater_T AC_WDAT28={JobModeId -187662529,ParamSetId -1375177600,CraterTime 0.100000,PostflowTime 0.100000,Channel1 30.0000,Channel2 1.00000,Channel3 0.0,Channel4 0.0,Channel5 0.0,Channel6 0.0,Channel7 0.0,Channel8 0.0,BurnBackTime 0.0}
DECL FDAT FP52={TOOL_NO 1,BASE_NO 0,IPO_FRAME #BASE,POINT2[] " ",TQ_STATE FALSE}
DECL LDAT LCPDAT15={ACC 100.000,APO_DIST 100.000,APO_FAC 50.0000,AXIS_VEL 100.000,AXIS_ACC 100.000,ORI_TYP #VAR,CIRC_TYP #BASE,JERK_FAC 50.0000,GEAR_JERK 50.0000,EXAX_IGN 0}
DECL E6POS XP52={X 1237.79492,Y -834.136475,Z 1624.22620,A -11.1505623,B -10.8155499,C 136.973816,S 2,T 10,E1 193.394,E2 193.959457,E3 193.454041,E4 0.0,E5 0.0,E6 0.0}
DECL E6POS XP53={X 1187.26587,Y -843.698853,Z 1664.27185,A -12.4819183,B -12.3824520,C 136.215851,S 2,T 10,E1 193.394,E2 193.959457,E3 193.454041,E4 0.0,E5 0.0,E6 0.0}
DECL FDAT FP53={TOOL_NO 1,BASE_NO 0,IPO_FRAME #BASE,POINT2[] " ",TQ_STATE FALSE}
DECL PDAT PPDAT40={VEL 100.000,ACC 100.000,APO_DIST 100.000,GEAR_JERK 50.0000,EXAX_IGN 3}
DECL ATBg_Start_T AS_WDAT29={JobModeId 1306102413,ParamSetId -1047099609,StartTime 0.0,PreFlowTime 0.0,Channel1 0.0,Channel2 2.00000,Channel3 0.0,Channel4 0.0,Channel5 0.0,Channel6 0.0,Channel7 0.0,Channel8 0.0,PurgeTime 0.0}
DECL ATBg_Weld_T AW_WDAT29={JobModeId -187662529,ParamSetId -430485013,Velocity 0.00830000,Channel1 30.0000,Channel2 1.00000,Channel3 0.0,Channel4 0.0,Channel5 0.0,Channel6 0.0,Channel7 0.0,Channel8 0.0}
DECL WTCg_WeaveDefinition_T WV_WDAT29={Pattern #None,Length 4.00000,Amplitude 2.00000,Angle 0.0}
DECL FDAT FP54={TOOL_NO 1,BASE_NO 0,IPO_FRAME #BASE,POINT2[] " ",TQ_STATE FALSE}
DECL PDAT PPDAT41={ACC 100.000,APO_DIST 100.000,APO_MODE #CPTP,GEAR_JERK 50.0000}
DECL E6POS XP54={X 1233.86,Y -871.477417,Z 1661.01746,A -17.3813877,B 8.68296,C -24.1851177,S 2,T 42,E1 193.394,E2 193.959457,E3 193.454041,E4 0.0,E5 0.0,E6 0.0}
DECL ATBg_Crater_T AC_WDAT30={JobModeId -187662529,ParamSetId -1375177600,CraterTime 0.100000,PostflowTime 0.100000,Channel1 30.0000,Channel2 1.00000,Channel3 0.0,Channel4 0.0,Channel5 0.0,Channel6 0.0,Channel7 0.0,Channel8 0.0,BurnBackTime 0.0}
DECL FDAT FP55={TOOL_NO 1,BASE_NO 0,IPO_FRAME #BASE,POINT2[] " ",TQ_STATE FALSE}
DECL LDAT LCPDAT16={ACC 100.000,APO_DIST 100.000,APO_FAC 50.0000,AXIS_VEL 100.000,AXIS_ACC 100.000,ORI_TYP #VAR,CIRC_TYP #BASE,JERK_FAC 50.0000,GEAR_JERK 50.0000,EXAX_IGN 0}
DECL E6POS XP55={X 1229.51489,Y -882.280884,Z 1661.04895,A -17.8144264,B 8.50245190,C -24.2574081,S 2,T 42,E1 193.394,E2 193.959457,E3 193.454041,E4 0.0,E5 0.0,E6 0.0}
DECL E6POS XP56={X 1198.65784,Y -856.923828,Z 1699.54797,A -17.8823528,B 7.26089811,C -24.7527294,S 2,T 42,E1 193.394,E2 193.959457,E3 193.454041,E4 0.0,E5 0.0,E6 0.0}
DECL FDAT FP56={TOOL_NO 1,BASE_NO 0,IPO_FRAME #BASE,POINT2[] " ",TQ_STATE FALSE}
DECL PDAT PPDAT42={VEL 100.000,ACC 100.000,APO_DIST 100.000,GEAR_JERK 50.0000,EXAX_IGN 3}
DECL ATBg_Start_T AS_WDAT31={JobModeId 1306102413,ParamSetId -1047099609,StartTime 0.0,PreFlowTime 0.0,Channel1 0.0,Channel2 2.00000,Channel3 0.0,Channel4 0.0,Channel5 0.0,Channel6 0.0,Channel7 0.0,Channel8 0.0,PurgeTime 0.0}
DECL ATBg_Weld_T AW_WDAT31={JobModeId -187662529,ParamSetId -430485013,Velocity 0.00830000,Channel1 30.0000,Channel2 1.00000,Channel3 0.0,Channel4 0.0,Channel5 0.0,Channel6 0.0,Channel7 0.0,Channel8 0.0}
DECL WTCg_WeaveDefinition_T WV_WDAT31={Pattern #None,Length 4.00000,Amplitude 2.00000,Angle 0.0}
DECL FDAT FP57={TOOL_NO 1,BASE_NO 0,IPO_FRAME #BASE,POINT2[] " ",TQ_STATE FALSE}
DECL PDAT PPDAT43={ACC 100.000,APO_DIST 100.000,APO_MODE #CPTP,GEAR_JERK 50.0000}
DECL E6POS XP57={X 1192.27454,Y -888.298523,Z 1498.37671,A -18.2437611,B 22.1260738,C -147.248505,S 0,T 42,E1 193.394,E2 193.959457,E3 193.454041,E4 0.0,E5 0.0,E6 0.0}
DECL ATBg_Crater_T AC_WDAT32={JobModeId -187662529,ParamSetId -1375177600,CraterTime 0.100000,PostflowTime 0.100000,Channel1 30.0000,Channel2 1.00000,Channel3 0.0,Channel4 0.0,Channel5 0.0,Channel6 0.0,Channel7 0.0,Channel8 0.0,BurnBackTime 0.0}
DECL FDAT FP58={TOOL_NO 1,BASE_NO 0,IPO_FRAME #BASE,POINT2[] " ",TQ_STATE FALSE}
DECL LDAT LCPDAT17={ACC 100.000,APO_DIST 100.000,APO_FAC 50.0000,AXIS_VEL 100.000,AXIS_ACC 100.000,ORI_TYP #VAR,CIRC_TYP #BASE,JERK_FAC 50.0000,GEAR_JERK 50.0000,EXAX_IGN 0}
DECL E6POS XP58={X 1180.67773,Y -900.955688,Z 1498.33386,A -18.7434597,B 23.0536861,C -146.821121,S 0,T 42,E1 193.394,E2 193.959457,E3 193.454041,E4 0.0,E5 0.0,E6 0.0}
DECL E6POS XP59={X 775.414917,Y -537.719116,Z 1950.34924,A -20.6824532,B 0.677307963,C -156.052979,S 0,T 42,E1 193.394,E2 193.959457,E3 193.454041,E4 0.0,E5 0.0,E6 0.0}
DECL FDAT FP59={TOOL_NO 1,BASE_NO 0,IPO_FRAME #BASE,POINT2[] " ",TQ_STATE FALSE}
DECL PDAT PPDAT44={VEL 100.000,ACC 100.000,APO_DIST 100.000,GEAR_JERK 50.0000,EXAX_IGN 3}
DECL E6POS XP60={X 775.414917,Y -537.719116,Z 1950.34924,A -20.6824532,B 0.677307963,C -156.052979,S 0,T 42,E1 39.2517242,E2 193.959457,E3 193.454041,E4 0.0,E5 0.0,E6 0.0}
DECL FDAT FP60={TOOL_NO 1,BASE_NO 0,IPO_FRAME #BASE,POINT2[] " ",TQ_STATE FALSE}
DECL PDAT PPDAT45={VEL 100.000,ACC 100.000,APO_DIST 100.000,GEAR_JERK 50.0000,EXAX_IGN 3}
DECL ATBg_Start_T AS_WDAT33={JobModeId 1306102413,ParamSetId -1047099609,StartTime 0.0,PreFlowTime 0.0,Channel1 0.0,Channel2 2.00000,Channel3 0.0,Channel4 0.0,Channel5 0.0,Channel6 0.0,Channel7 0.0,Channel8 0.0,PurgeTime 0.0}
DECL ATBg_Weld_T AW_WDAT33={JobModeId -187662529,ParamSetId -430485013,Velocity 0.00830000,Channel1 30.0000,Channel2 1.00000,Channel3 0.0,Channel4 0.0,Channel5 0.0,Channel6 0.0,Channel7 0.0,Channel8 0.0}
DECL WTCg_WeaveDefinition_T WV_WDAT33={Pattern #None,Length 4.00000,Amplitude 2.00000,Angle 0.0}
DECL FDAT FP61={TOOL_NO 1,BASE_NO 0,IPO_FRAME #BASE,POINT2[] " ",TQ_STATE FALSE}
DECL PDAT PPDAT46={ACC 100.000,APO_DIST 100.000,APO_MODE #CPTP,GEAR_JERK 50.0000}
DECL E6POS XP61={X 1264.14771,Y -888.481079,Z 1526.40186,A 3.01134205,B 15.7321072,C 103.378540,S 2,T 42,E1 63.9584122,E2 193.959412,E3 193.453964,E4 0.0,E5 0.0,E6 0.0}
DECL ATBg_Crater_T AC_WDAT34={JobModeId -187662529,ParamSetId -1375177600,CraterTime 0.100000,PostflowTime 0.100000,Channel1 30.0000,Channel2 1.00000,Channel3 0.0,Channel4 0.0,Channel5 0.0,Channel6 0.0,Channel7 0.0,Channel8 0.0,BurnBackTime 0.0}
DECL FDAT FP62={TOOL_NO 1,BASE_NO 0,IPO_FRAME #BASE,POINT2[] " ",TQ_STATE FALSE}
DECL LDAT LCPDAT18={ACC 100.000,APO_DIST 100.000,APO_FAC 50.0000,AXIS_VEL 100.000,AXIS_ACC 100.000,ORI_TYP #VAR,CIRC_TYP #BASE,JERK_FAC 50.0000,GEAR_JERK 50.0000,EXAX_IGN 0}
DECL E6POS XP62={X 1266.80566,Y -885.966064,Z 1520.92126,A 3.57900286,B 16.3062973,C 104.266014,S 2,T 42,E1 63.9584465,E2 193.959412,E3 193.453964,E4 0.0,E5 0.0,E6 0.0}
DECL ATBg_Start_T AS_WDAT35={JobModeId 1306102413,ParamSetId -1047099609,StartTime 0.0,PreFlowTime 0.0,Channel1 0.0,Channel2 2.00000,Channel3 0.0,Channel4 0.0,Channel5 0.0,Channel6 0.0,Channel7 0.0,Channel8 0.0,PurgeTime 0.0}
DECL ATBg_Weld_T AW_WDAT35={JobModeId -187662529,ParamSetId -430485013,Velocity 0.00830000,Channel1 30.0000,Channel2 1.00000,Channel3 0.0,Channel4 0.0,Channel5 0.0,Channel6 0.0,Channel7 0.0,Channel8 0.0}
DECL WTCg_WeaveDefinition_T WV_WDAT35={Pattern #None,Length 4.00000,Amplitude 2.00000,Angle 0.0}
DECL FDAT FP63={TOOL_NO 1,BASE_NO 0,IPO_FRAME #BASE,POINT2[] " ",TQ_STATE FALSE}
DECL PDAT PPDAT47={ACC 100.000,APO_DIST 100.000,APO_MODE #CPTP,GEAR_JERK 50.0000}
DECL E6POS XP63={X 1378.29102,Y -638.791870,Z 1512.36633,A 15.4253092,B 20.5481892,C 99.7943726,S 2,T 42,E1 63.9585266,E2 193.959412,E3 193.453964,E4 0.0,E5 0.0,E6 0.0}
DECL ATBg_Crater_T AC_WDAT36={JobModeId -187662529,ParamSetId -1375177600,CraterTime 0.100000,PostflowTime 0.100000,Channel1 30.0000,Channel2 1.00000,Channel3 0.0,Channel4 0.0,Channel5 0.0,Channel6 0.0,Channel7 0.0,Channel8 0.0,BurnBackTime 0.0}
DECL FDAT FP64={TOOL_NO 1,BASE_NO 0,IPO_FRAME #BASE,POINT2[] " ",TQ_STATE FALSE}
DECL LDAT LCPDAT19={ACC 100.000,APO_DIST 100.000,APO_FAC 50.0000,AXIS_VEL 100.000,AXIS_ACC 100.000,ORI_TYP #VAR,CIRC_TYP #BASE,JERK_FAC 50.0000,GEAR_JERK 50.0000,EXAX_IGN 0}
DECL E6POS XP64={X 1373.91870,Y -654.769104,Z 1511.57153,A 14.8009529,B 20.4592934,C 99.4732513,S 2,T 42,E1 63.9585266,E2 193.959412,E3 193.453964,E4 0.0,E5 0.0,E6 0.0}
DECL ATBg_Start_T AS_WDAT37={JobModeId 1306102413,ParamSetId -1047099609,StartTime 0.0,PreFlowTime 0.0,Channel1 0.0,Channel2 2.00000,Channel3 0.0,Channel4 0.0,Channel5 0.0,Channel6 0.0,Channel7 0.0,Channel8 0.0,PurgeTime 0.0}
DECL ATBg_Weld_T AW_WDAT37={JobModeId -187662529,ParamSetId -430485013,Velocity 0.00830000,Channel1 30.0000,Channel2 1.00000,Channel3 0.0,Channel4 0.0,Channel5 0.0,Channel6 0.0,Channel7 0.0,Channel8 0.0}
DECL WTCg_WeaveDefinition_T WV_WDAT37={Pattern #None,Length 4.00000,Amplitude 2.00000,Angle 0.0}
DECL FDAT FP65={TOOL_NO 1,BASE_NO 0,IPO_FRAME #BASE,POINT2[] " ",TQ_STATE FALSE}
DECL PDAT PPDAT48={ACC 100.000,APO_DIST 100.000,APO_MODE #CPTP,GEAR_JERK 50.0000}
DECL E6POS XP65={X 1467.26331,Y -272.376038,Z 1535.07397,A 29.8293266,B 19.9220467,C 85.8883896,S 2,T 42,E1 63.9585266,E2 193.959412,E3 193.453964,E4 0.0,E5 0.0,E6 0.0}
DECL ATBg_Crater_T AC_WDAT38={JobModeId -187662529,ParamSetId -1375177600,CraterTime 0.100000,PostflowTime 0.100000,Channel1 30.0000,Channel2 1.00000,Channel3 0.0,Channel4 0.0,Channel5 0.0,Channel6 0.0,Channel7 0.0,Channel8 0.0,BurnBackTime 0.0}
DECL FDAT FP66={TOOL_NO 1,BASE_NO 0,IPO_FRAME #BASE,POINT2[] " ",TQ_STATE FALSE}
DECL LDAT LCPDAT20={ACC 100.000,APO_DIST 100.000,APO_FAC 50.0000,AXIS_VEL 100.000,AXIS_ACC 100.000,ORI_TYP #VAR,CIRC_TYP #BASE,JERK_FAC 50.0000,GEAR_JERK 50.0000,EXAX_IGN 0}
DECL E6POS XP66={X 1467.65417,Y -283.093353,Z 1532.97620,A 29.4471760,B 19.9605255,C 85.9277496,S 2,T 42,E1 63.9585266,E2 193.959412,E3 193.453964,E4 0.0,E5 0.0,E6 0.0}
DECL ATBg_Start_T AS_WDAT39={JobModeId 1306102413,ParamSetId -1047099609,StartTime 0.0,PreFlowTime 0.0,Channel1 0.0,Channel2 2.00000,Channel3 0.0,Channel4 0.0,Channel5 0.0,Channel6 0.0,Channel7 0.0,Channel8 0.0,PurgeTime 0.0}
DECL ATBg_Weld_T AW_WDAT39={JobModeId -187662529,ParamSetId -430485013,Velocity 0.00830000,Channel1 30.0000,Channel2 1.00000,Channel3 0.0,Channel4 0.0,Channel5 0.0,Channel6 0.0,Channel7 0.0,Channel8 0.0}
DECL WTCg_WeaveDefinition_T WV_WDAT39={Pattern #None,Length 4.00000,Amplitude 2.00000,Angle 0.0}
DECL FDAT FP67={TOOL_NO 1,BASE_NO 0,IPO_FRAME #BASE,POINT2[] " ",TQ_STATE FALSE}
DECL PDAT PPDAT49={ACC 100.000,APO_DIST 100.000,APO_MODE #CPTP,GEAR_JERK 50.0000}
DECL E6POS XP67={X 1518.96875,Y -34.1009827,Z 1505.96338,A 46.2905922,B 23.6734219,C 71.8355408,S 2,T 42,E1 63.9585266,E2 193.959412,E3 193.453964,E4 0.0,E5 0.0,E6 0.0}
DECL ATBg_Crater_T AC_WDAT40={JobModeId -187662529,ParamSetId -1375177600,CraterTime 0.100000,PostflowTime 0.100000,Channel1 30.0000,Channel2 1.00000,Channel3 0.0,Channel4 0.0,Channel5 0.0,Channel6 0.0,Channel7 0.0,Channel8 0.0,BurnBackTime 0.0}
DECL FDAT FP68={TOOL_NO 1,BASE_NO 0,IPO_FRAME #BASE,POINT2[] " ",TQ_STATE FALSE}
DECL LDAT LCPDAT21={ACC 100.000,APO_DIST 100.000,APO_FAC 50.0000,AXIS_VEL 100.000,AXIS_ACC 100.000,ORI_TYP #VAR,CIRC_TYP #BASE,JERK_FAC 50.0000,GEAR_JERK 50.0000,EXAX_IGN 0}
DECL E6POS XP68={X 1520.88782,Y -15.9589958,Z 1505.16199,A 46.9704819,B 23.6559772,C 71.8110886,S 2,T 42,E1 63.9585266,E2 193.959412,E3 193.453964,E4 0.0,E5 0.0,E6 0.0}
DECL ATBg_Start_T AS_WDAT41={JobModeId 1306102413,ParamSetId -1047099609,StartTime 0.0,PreFlowTime 0.0,Channel1 0.0,Channel2 2.00000,Channel3 0.0,Channel4 0.0,Channel5 0.0,Channel6 0.0,Channel7 0.0,Channel8 0.0,PurgeTime 0.0}
DECL ATBg_Weld_T AW_WDAT41={JobModeId -187662529,ParamSetId -430485013,Velocity 0.00830000,Channel1 30.0000,Channel2 1.00000,Channel3 0.0,Channel4 0.0,Channel5 0.0,Channel6 0.0,Channel7 0.0,Channel8 0.0}
DECL WTCg_WeaveDefinition_T WV_WDAT41={Pattern #None,Length 4.00000,Amplitude 2.00000,Angle 0.0}
DECL FDAT FP69={TOOL_NO 1,BASE_NO 0,IPO_FRAME #BASE,POINT2[] " ",TQ_STATE FALSE}
DECL PDAT PPDAT50={ACC 100.000,APO_DIST 100.000,APO_MODE #CPTP,GEAR_JERK 50.0000}
DECL E6POS XP69={X 1482.85425,Y 344.327789,Z 1555.15930,A 53.9943581,B 17.9291592,C 69.6620865,S 2,T 43,E1 63.9585266,E2 193.959412,E3 193.453964,E4 0.0,E5 0.0,E6 0.0}
DECL ATBg_Crater_T AC_WDAT42={JobModeId -187662529,ParamSetId -1375177600,CraterTime 0.100000,PostflowTime 0.100000,Channel1 30.0000,Channel2 1.00000,Channel3 0.0,Channel4 0.0,Channel5 0.0,Channel6 0.0,Channel7 0.0,Channel8 0.0,BurnBackTime 0.0}
DECL FDAT FP70={TOOL_NO 1,BASE_NO 0,IPO_FRAME #BASE,POINT2[] " ",TQ_STATE FALSE}
DECL LDAT LCPDAT22={ACC 100.000,APO_DIST 100.000,APO_FAC 50.0000,AXIS_VEL 100.000,AXIS_ACC 100.000,ORI_TYP #VAR,CIRC_TYP #BASE,JERK_FAC 50.0000,GEAR_JERK 50.0000,EXAX_IGN 0}
DECL E6POS XP70={X 1479.48779,Y 364.142761,Z 1556.53235,A 54.7018547,B 17.7712841,C 69.4979,S 2,T 43,E1 63.9585266,E2 193.959412,E3 193.453964,E4 0.0,E5 0.0,E6 0.0}
DECL E6POS XP71={X 994.901,Y 278.536743,Z 1945.18140,A 52.2360458,B 4.75616121,C 57.0029526,S 2,T 43,E1 63.9585266,E2 193.959412,E3 193.453964,E4 0.0,E5 0.0,E6 0.0}
DECL FDAT FP71={TOOL_NO 1,BASE_NO 0,IPO_FRAME #BASE,POINT2[] " ",TQ_STATE FALSE}
DECL PDAT PPDAT51={VEL 100.000,ACC 100.000,APO_DIST 100.000,GEAR_JERK 50.0000,EXAX_IGN 3}
DECL ATBg_Start_T AS_WDAT43={JobModeId 1306102413,ParamSetId -1047099609,StartTime 0.0,PreFlowTime 0.0,Channel1 0.0,Channel2 2.00000,Channel3 0.0,Channel4 0.0,Channel5 0.0,Channel6 0.0,Channel7 0.0,Channel8 0.0,PurgeTime 0.0}
DECL ATBg_Weld_T AW_WDAT43={JobModeId -187662529,ParamSetId -430485013,Velocity 0.00830000,Channel1 30.0000,Channel2 1.00000,Channel3 0.0,Channel4 0.0,Channel5 0.0,Channel6 0.0,Channel7 0.0,Channel8 0.0}
DECL WTCg_WeaveDefinition_T WV_WDAT43={Pattern #None,Length 4.00000,Amplitude 2.00000,Angle 0.0}
DECL FDAT FP72={TOOL_NO 1,BASE_NO 0,IPO_FRAME #BASE,POINT2[] " ",TQ_STATE FALSE}
DECL PDAT PPDAT52={ACC 100.000,APO_DIST 100.000,APO_MODE #CPTP,GEAR_JERK 50.0000}
DECL E6POS XP72={X 1419.64844,Y 379.711395,Z 1619.32703,A 44.0833893,B -10.5155697,C 98.5163193,S 2,T 43,E1 -0.571967244,E2 193.829330,E3 193.453964,E4 0.0,E5 0.0,E6 0.0}
DECL ATBg_Crater_T AC_WDAT44={JobModeId -187662529,ParamSetId -1375177600,CraterTime 0.100000,PostflowTime 0.100000,Channel1 30.0000,Channel2 1.00000,Channel3 0.0,Channel4 0.0,Channel5 0.0,Channel6 0.0,Channel7 0.0,Channel8 0.0,BurnBackTime 0.0}
DECL FDAT FP73={TOOL_NO 1,BASE_NO 0,IPO_FRAME #BASE,POINT2[] " ",TQ_STATE FALSE}
DECL LDAT LCPDAT23={ACC 100.000,APO_DIST 100.000,APO_FAC 50.0000,AXIS_VEL 100.000,AXIS_ACC 100.000,ORI_TYP #VAR,CIRC_TYP #BASE,JERK_FAC 50.0000,GEAR_JERK 50.0000,EXAX_IGN 0}
DECL E6POS XP73={X 1423.85510,Y 361.552246,Z 1617.04346,A 43.3382950,B -10.3582993,C 98.6139526,S 2,T 43,E1 -0.571967244,E2 193.829330,E3 193.453964,E4 0.0,E5 0.0,E6 0.0}
DECL E6POS XP74={X 1237.78,Y 322.197296,Z 1801.70483,A 44.4825630,B -17.6892014,C 93.9040451,S 2,T 43,E1 -0.571967244,E2 193.829330,E3 193.453964,E4 0.0,E5 0.0,E6 0.0}
DECL FDAT FP74={TOOL_NO 1,BASE_NO 0,IPO_FRAME #BASE,POINT2[] " ",TQ_STATE FALSE}
DECL PDAT PPDAT53={VEL 100.000,ACC 100.000,APO_DIST 100.000,GEAR_JERK 50.0000,EXAX_IGN 3}
DECL ATBg_Start_T AS_WDAT45={JobModeId 1306102413,ParamSetId -1047099609,StartTime 0.0,PreFlowTime 0.0,Channel1 0.0,Channel2 2.00000,Channel3 0.0,Channel4 0.0,Channel5 0.0,Channel6 0.0,Channel7 0.0,Channel8 0.0,PurgeTime 0.0}
DECL ATBg_Weld_T AW_WDAT45={JobModeId -187662529,ParamSetId -430485013,Velocity 0.00830000,Channel1 30.0000,Channel2 1.00000,Channel3 0.0,Channel4 0.0,Channel5 0.0,Channel6 0.0,Channel7 0.0,Channel8 0.0}
DECL WTCg_WeaveDefinition_T WV_WDAT45={Pattern #None,Length 4.00000,Amplitude 2.00000,Angle 0.0}
DECL FDAT FP75={TOOL_NO 1,BASE_NO 0,IPO_FRAME #BASE,POINT2[] " ",TQ_STATE FALSE}
DECL PDAT PPDAT54={ACC 100.000,APO_DIST 100.000,APO_MODE #CPTP,GEAR_JERK 50.0000}
DECL E6POS XP75={X 1447.43835,Y 22.4731827,Z 1600.42542,A 34.4591331,B -2.99060321,C 90.7398300,S 2,T 42,E1 -0.571967244,E2 193.829330,E3 193.453964,E4 0.0,E5 0.0,E6 0.0}
DECL ATBg_Crater_T AC_WDAT46={JobModeId -187662529,ParamSetId -1375177600,CraterTime 0.100000,PostflowTime 0.100000,Channel1 30.0000,Channel2 1.00000,Channel3 0.0,Channel4 0.0,Channel5 0.0,Channel6 0.0,Channel7 0.0,Channel8 0.0,BurnBackTime 0.0}
DECL FDAT FP76={TOOL_NO 1,BASE_NO 0,IPO_FRAME #BASE,POINT2[] " ",TQ_STATE FALSE}
DECL LDAT LCPDAT24={ACC 100.000,APO_DIST 100.000,APO_FAC 50.0000,AXIS_VEL 100.000,AXIS_ACC 100.000,ORI_TYP #VAR,CIRC_TYP #BASE,JERK_FAC 50.0000,GEAR_JERK 50.0000,EXAX_IGN 0}
DECL E6POS XP76={X 1447.68677,Y 4.22323036,Z 1598.95911,A 33.7338181,B -2.90925980,C 90.8003540,S 2,T 42,E1 -0.571967244,E2 193.829330,E3 193.453964,E4 0.0,E5 0.0,E6 0.0}
DECL E6POS XP77={X 1384.67957,Y 7.39358425,Z 1666.38965,A 33.8657913,B -5.35998583,C 88.9704819,S 2,T 42,E1 -0.571967244,E2 193.829330,E3 193.453964,E4 0.0,E5 0.0,E6 0.0}
DECL FDAT FP77={TOOL_NO 1,BASE_NO 0,IPO_FRAME #BASE,POINT2[] " ",TQ_STATE FALSE}
DECL PDAT PPDAT55={VEL 100.000,ACC 100.000,APO_DIST 100.000,GEAR_JERK 50.0000,EXAX_IGN 3}
DECL ATBg_Start_T AS_WDAT47={JobModeId 1306102413,ParamSetId -1047099609,StartTime 0.0,PreFlowTime 0.0,Channel1 0.0,Channel2 2.00000,Channel3 0.0,Channel4 0.0,Channel5 0.0,Channel6 0.0,Channel7 0.0,Channel8 0.0,PurgeTime 0.0}
DECL ATBg_Weld_T AW_WDAT47={JobModeId -187662529,ParamSetId -430485013,Velocity 0.00830000,Channel1 30.0000,Channel2 1.00000,Channel3 0.0,Channel4 0.0,Channel5 0.0,Channel6 0.0,Channel7 0.0,Channel8 0.0}
DECL WTCg_WeaveDefinition_T WV_WDAT47={Pattern #None,Length 4.00000,Amplitude 2.00000,Angle 0.0}
DECL FDAT FP78={TOOL_NO 1,BASE_NO 0,IPO_FRAME #BASE,POINT2[] " ",TQ_STATE FALSE}
DECL PDAT PPDAT56={ACC 100.000,APO_DIST 100.000,APO_MODE #CPTP,GEAR_JERK 50.0000}
DECL E6POS XP78={X 1420.44470,Y -260.332886,Z 1594.88318,A 23.0712452,B -2.55928659,C 93.0881653,S 2,T 42,E1 -0.571967244,E2 193.829330,E3 193.453964,E4 0.0,E5 0.0,E6 0.0}
DECL ATBg_Crater_T AC_WDAT48={JobModeId -187662529,ParamSetId -1375177600,CraterTime 0.100000,PostflowTime 0.100000,Channel1 30.0000,Channel2 1.00000,Channel3 0.0,Channel4 0.0,Channel5 0.0,Channel6 0.0,Channel7 0.0,Channel8 0.0,BurnBackTime 0.0}
DECL FDAT FP79={TOOL_NO 1,BASE_NO 0,IPO_FRAME #BASE,POINT2[] " ",TQ_STATE FALSE}
DECL LDAT LCPDAT25={ACC 100.000,APO_DIST 100.000,APO_FAC 50.0000,AXIS_VEL 100.000,AXIS_ACC 100.000,ORI_TYP #VAR,CIRC_TYP #BASE,JERK_FAC 50.0000,GEAR_JERK 50.0000,EXAX_IGN 0}
DECL E6POS XP79={X 1418.97449,Y -282.628448,Z 1596.02136,A 22.3030128,B -2.72646022,C 90.7286,S 2,T 42,E1 -0.571967244,E2 193.829330,E3 193.453964,E4 0.0,E5 0.0,E6 0.0}
DECL E6POS XP80={X 1220.08362,Y -560.013550,Z 1746.04102,A 14.0401382,B -1.45351505,C 59.8836098,S 2,T 42,E1 -0.571967244,E2 193.829330,E3 193.453964,E4 0.0,E5 0.0,E6 0.0}
DECL FDAT FP80={TOOL_NO 1,BASE_NO 0,IPO_FRAME #BASE,POINT2[] " ",TQ_STATE FALSE}
DECL PDAT PPDAT57={VEL 100.000,ACC 100.000,APO_DIST 100.000,GEAR_JERK 50.0000,EXAX_IGN 3}
DECL ATBg_Start_T AS_WDAT49={JobModeId 1306102413,ParamSetId -1047099609,StartTime 0.0,PreFlowTime 0.0,Channel1 0.0,Channel2 2.00000,Channel3 0.0,Channel4 0.0,Channel5 0.0,Channel6 0.0,Channel7 0.0,Channel8 0.0,PurgeTime 0.0}
DECL ATBg_Weld_T AW_WDAT49={JobModeId -187662529,ParamSetId -430485013,Velocity 0.00830000,Channel1 30.0000,Channel2 1.00000,Channel3 0.0,Channel4 0.0,Channel5 0.0,Channel6 0.0,Channel7 0.0,Channel8 0.0}
DECL WTCg_WeaveDefinition_T WV_WDAT49={Pattern #None,Length 4.00000,Amplitude 2.00000,Angle 0.0}
DECL FDAT FP81={TOOL_NO 1,BASE_NO 0,IPO_FRAME #BASE,POINT2[] " ",TQ_STATE FALSE}
DECL PDAT PPDAT58={ACC 100.000,APO_DIST 100.000,APO_MODE #CPTP,GEAR_JERK 50.0000}
DECL E6POS XP81={X 1354.26074,Y -634.417053,Z 1589.40454,A 14.1318378,B 3.65171266,C 64.6567154,S 2,T 42,E1 -0.571967244,E2 193.829330,E3 193.453964,E4 0.0,E5 0.0,E6 0.0}
DECL ATBg_Crater_T AC_WDAT50={JobModeId -187662529,ParamSetId -1375177600,CraterTime 0.100000,PostflowTime 0.100000,Channel1 30.0000,Channel2 1.00000,Channel3 0.0,Channel4 0.0,Channel5 0.0,Channel6 0.0,Channel7 0.0,Channel8 0.0,BurnBackTime 0.0}
DECL FDAT FP82={TOOL_NO 1,BASE_NO 0,IPO_FRAME #BASE,POINT2[] " ",TQ_STATE FALSE}
DECL LDAT LCPDAT26={ACC 100.000,APO_DIST 100.000,APO_FAC 50.0000,AXIS_VEL 100.000,AXIS_ACC 100.000,ORI_TYP #VAR,CIRC_TYP #BASE,JERK_FAC 50.0000,GEAR_JERK 50.0000,EXAX_IGN 0}
DECL E6POS XP82={X 1352.78101,Y -660.651367,Z 1580.30505,A 14.4475975,B 4.36072063,C 64.7877121,S 2,T 42,E1 -0.571967244,E2 193.829330,E3 193.453964,E4 0.0,E5 0.0,E6 0.0}
DECL E6POS XP83={X 1271.57,Y -613.565796,Z 1683.91687,A 14.2951546,B 1.11499119,C 61.5984039,S 2,T 42,E1 -0.571967244,E2 193.829330,E3 193.453964,E4 0.0,E5 0.0,E6 0.0}
DECL FDAT FP83={TOOL_NO 1,BASE_NO 0,IPO_FRAME #BASE,POINT2[] " ",TQ_STATE FALSE}
DECL PDAT PPDAT59={VEL 100.000,ACC 100.000,APO_DIST 100.000,GEAR_JERK 50.0000,EXAX_IGN 3}
DECL ATBg_Start_T AS_WDAT51={JobModeId 1306102413,ParamSetId -1047099609,StartTime 0.0,PreFlowTime 0.0,Channel1 0.0,Channel2 2.00000,Channel3 0.0,Channel4 0.0,Channel5 0.0,Channel6 0.0,Channel7 0.0,Channel8 0.0,PurgeTime 0.0}
DECL ATBg_Weld_T AW_WDAT51={JobModeId -187662529,ParamSetId -430485013,Velocity 0.00830000,Channel1 30.0000,Channel2 1.00000,Channel3 0.0,Channel4 0.0,Channel5 0.0,Channel6 0.0,Channel7 0.0,Channel8 0.0}
DECL WTCg_WeaveDefinition_T WV_WDAT51={Pattern #None,Length 4.00000,Amplitude 2.00000,Angle 0.0}
DECL FDAT FP84={TOOL_NO 1,BASE_NO 0,IPO_FRAME #BASE,POINT2[] " ",TQ_STATE FALSE}
DECL PDAT PPDAT60={ACC 100.000,APO_DIST 100.000,APO_MODE #CPTP,GEAR_JERK 50.0000}
DECL E6POS XP84={X 1270.70068,Y -931.227539,Z 1509.36133,A 14.6498194,B 10.0588856,C 79.5254288,S 2,T 42,E1 -0.571961224,E2 193.829300,E3 193.453918,E4 0.0,E5 0.0,E6 0.0}
DECL ATBg_Crater_T AC_WDAT52={JobModeId -187662529,ParamSetId -1375177600,CraterTime 0.100000,PostflowTime 0.100000,Channel1 30.0000,Channel2 1.00000,Channel3 0.0,Channel4 0.0,Channel5 0.0,Channel6 0.0,Channel7 0.0,Channel8 0.0,BurnBackTime 0.0}
DECL FDAT FP85={TOOL_NO 1,BASE_NO 0,IPO_FRAME #BASE,POINT2[] " ",TQ_STATE FALSE}
DECL LDAT LCPDAT27={ACC 100.000,APO_DIST 100.000,APO_FAC 50.0000,AXIS_VEL 100.000,AXIS_ACC 100.000,ORI_TYP #VAR,CIRC_TYP #BASE,JERK_FAC 50.0000,GEAR_JERK 50.0000,EXAX_IGN 0}
DECL E6POS XP85={X 1264.23535,Y -948.284241,Z 1507.87646,A 13.9848785,B 9.89103699,C 79.2727432,S 2,T 42,E1 -0.571961224,E2 193.829300,E3 193.453918,E4 0.0,E5 0.0,E6 0.0}
DECL E6POS XP86={X 1033.11694,Y -740.220154,Z 1831.33533,A 12.7748480,B 1.60397112,C 67.2652,S 2,T 42,E1 -0.571961224,E2 193.829300,E3 193.453918,E4 0.0,E5 0.0,E6 0.0}
DECL FDAT FP86={TOOL_NO 1,BASE_NO 0,IPO_FRAME #BASE,POINT2[] " ",TQ_STATE FALSE}
DECL PDAT PPDAT61={VEL 100.000,ACC 100.000,APO_DIST 100.000,GEAR_JERK 50.0000,EXAX_IGN 3}
DECL E6POS XP87={X 802.714966,Y -628.910278,Z 1971.60498,A -15.5495539,B -26.0840855,C 130.575607,S 2,T 10,E1 193.394,E2 193.959457,E3 193.454041,E4 0.0,E5 0.0,E6 0.0}
DECL FDAT FP87={TOOL_NO 1,BASE_NO 0,IPO_FRAME #BASE,POINT2[] " ",TQ_STATE FALSE}
